KUKA KRL program: MyProgram_262().src

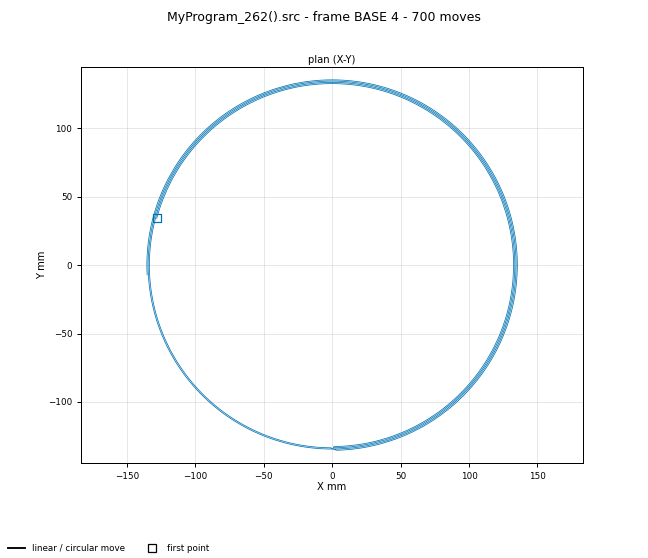
[picture p0: tool path of MyProgram_262().src in frame BASE 4, 700 of 700 moves have a stored position in this frame; points joined in program order, loops and branches not executed]
&ACCESS RVP
&REL 1
&PARAM TEMPLATE = C:\KRC\Roboter\Template\vorgabe
&PARAM EDITMASK = *
DEF MyProgram_262()
; ---- Setting reference (Base) ----
$BASE = BASE_DATA[4]

; --------------------------
; ---- Setting tool (TCP) ----
$TOOL = TOOL_DATA[3]
; --------------------------

$VEL.CP = VEL_APROX_PRINT
Startdeposition()
$VEL.CP = VEL_PRINT
LIN {X -128.1106,Y 34.116,Z 168,A 165.358,B 10.6516,C 0.1235,E1 10.4979,E2 285.5188} C_DIS
LIN {X -127.1106,Y 37.6736,Z 168,A 163.7129,B 10.6516,C 0.1199,E1 10.4991,E2 287.1678} C_DIS
LIN {X -125.942,Y 41.4132,Z 168,A 161.9508,B 10.6516,C 0.1164,E1 10.5006,E2 288.9361} C_DIS
LIN {X -124.5968,Y 45.2984,Z 168,A 160.2681,B 10.6518,C 0.1097,E1 10.5022,E2 290.6058} C_DIS
LIN {X -123.3963,Y 48.4742,Z 168,A 158.6213,B 10.6518,C 0.109,E1 10.5039,E2 292.272} C_DIS
LIN {X -120.4612,Y 55.3657,Z 168,A 155.2422,B 10.6518,C 0.1029,E1 10.5077,E2 295.6641} C_DIS
LIN {X -117.7741,Y 60.8777,Z 168,A 152.6518,B 10.6518,C 0.0948,E1 10.5109,E2 298.2447} C_DIS
LIN {X -115.8376,Y 64.4859,Z 168,A 150.9654,B 10.6519,C 0.0886,E1 10.5131,E2 299.9194} C_DIS
LIN {X -113.7435,Y 68.1115,Z 168,A 149.1743,B 10.6519,C 0.0836,E1 10.5157,E2 301.7063} C_DIS
LIN {X -110.9155,Y 72.626,Z 168,A 147.0442,B 10.6521,C 0.0746,E1 10.5188,E2 303.8138} C_DIS
LIN {X -109.3081,Y 75.0228,Z 168,A 145.5131,B 10.6521,C 0.0769,E1 10.5213,E2 305.3767} C_DIS
LIN {X -106.8216,Y 78.5228,Z 168,A 143.6005,B 10.6521,C 0.0735,E1 10.5244,E2 307.294} C_DIS
LIN {X -104.1665,Y 82.0125,Z 168,A 141.7197,B 10.6521,C 0.0688,E1 10.5276,E2 309.1711} C_DIS
LIN {X -101.3729,Y 85.4419,Z 168,A 139.7836,B 10.6521,C 0.0649,E1 10.531,E2 311.1079} C_DIS
LIN {X -98.5887,Y 88.6398,Z 168,A 137.9057,B 10.6521,C 0.0617,E1 10.5345,E2 312.9892} C_DIS
LIN {X -95.5472,Y 91.9108,Z 168,A 135.9314,B 10.6521,C 0.0583,E1 10.5383,E2 314.9666} C_DIS
LIN {X -92.4629,Y 95.0127,Z 168,A 134.0224,B 10.6521,C 0.0547,E1 10.5421,E2 316.8759} C_DIS
LIN {X -89.2719,Y 98.0167,Z 168,A 132.1098,B 10.6521,C 0.0512,E1 10.546,E2 318.7886} C_DIS
LIN {X -86.0227,Y 100.8802,Z 168,A 130.2329,B 10.6522,C 0.0477,E1 10.55,E2 320.6642} C_DIS
LIN {X -82.589,Y 103.7099,Z 168,A 128.2998,B 10.6522,C 0.0443,E1 10.5542,E2 322.5966} C_DIS
LIN {X -79.0187,Y 106.4555,Z 168,A 126.3454,B 10.6522,C 0.0409,E1 10.5585,E2 324.55} C_DIS
LIN {X -75.68,Y 108.8542,Z 168,A 124.5397,B 10.6522,C 0.0384,E1 10.5626,E2 326.3574} C_DIS
LIN {X -72.0548,Y 111.2871,Z 168,A 122.6403,B 10.6522,C 0.0355,E1 10.5671,E2 328.2565} C_DIS
LIN {X -68.5115,Y 113.5028,Z 168,A 120.4154,B 10.6522,C 0.041,E1 10.5725,E2 330.5284} C_DIS
LIN {X -64.82,Y 115.6507,Z 168,A 118.4323,B 10.6522,C 0.041,E1 10.5774,E2 332.5256} C_DIS
LIN {X -60.5627,Y 117.9344,Z 168,A 117.1036,B 10.6522,C 0.0229,E1 10.5804,E2 333.7644} C_DIS
LIN {X -53.8546,Y 121.1443,Z 168,A 113.7444,B 10.6522,C 0.0217,E1 10.589,E2 337.1379} C_DIS
LIN {X -50.7874,Y 122.4619,Z 168,A 112.2996,B 10.6522,C 0.02,E1 10.5927,E2 338.5818} C_DIS
LIN {X -47.6217,Y 123.7277,Z 168,A 110.7107,B 10.6522,C 0.0207,E1 10.5968,E2 340.183} C_DIS
LIN {X -43.62,Y 125.194,Z 168,A 108.8903,B 10.6522,C 0.0184,E1 10.6016,E2 341.9994} C_DIS
LIN {X -37.8929,Y 127.0464,Z 168,A 106.3941,B 10.6523,C 0.0138,E1 10.6082,E2 344.4815} C_DIS
LIN {X -34.225,Y 128.0815,Z 168,A 104.6813,B 10.6523,C 0.0138,E1 10.6128,E2 346.2008} C_DIS
LIN {X -31.0238,Y 128.8943,Z 168,A 102.7778,B 10.6523,C 0.0227,E1 10.6181,E2 348.1586} C_DIS
LIN {X -26.9831,Y 129.8016,Z 168,A 101.3362,B 10.6523,C 0.0143,E1 10.622,E2 349.5587} C_DIS
LIN {X -23.2949,Y 130.5128,Z 168,A 99.8078,B 10.6523,C 0.0113,E1 10.6261,E2 351.075} C_DIS
LIN {X -20.1004,Y 131.043,Z 168,A 98.4194,B 10.6523,C 0.0104,E1 10.63,E2 352.4612} C_DIS
LIN {X -16.8033,Y 131.507,Z 168,A 96.8595,B 10.6523,C 0.0123,E1 10.6343,E2 354.0344} C_DIS
LIN {X -12.6917,Y 131.9667,Z 168,A 95.1681,B 10.6523,C 0.0096,E1 10.639,E2 355.7135} C_DIS
LIN {X -9.1067,Y 132.2636,Z 168,A 93.5018,B 10.6523,C 0.0116,E1 10.6436,E2 357.392} C_DIS
LIN {X -5.0768,Y 132.4784,Z 168,A 91.8892,B 10.6523,C 0.0085,E1 10.6481,E2 358.9883} C_DIS
LIN {X -1.0548,Y 132.5719,Z 168,A 90.0932,B 10.6523,C 0.0096,E1 10.6531,E2 360.7902} C_DIS
LIN {X 3.0141,Y 132.5431,Z 168,A 88.2853,B 10.6523,C 0.0106,E1 10.6582,E2 362.6032} C_DIS
LIN {X 6.8789,Y 132.3972,Z 168,A 86.621,B 10.6523,C 0.0106,E1 10.6628,E2 364.2659} C_DIS
LIN {X 11.0997,Y 132.1101,Z 168,A 84.8958,B 10.6523,C 0.0087,E1 10.6676,E2 365.9783} C_DIS
LIN {X 14.6757,Y 131.7617,Z 168,A 83.2175,B 10.6523,C 0.0118,E1 10.6723,E2 367.6707} C_DIS
LIN {X 18.6908,Y 131.2514,Z 168,A 81.5841,B 10.6523,C 0.0099,E1 10.6768,E2 369.29} C_DIS
LIN {X 22.2463,Y 130.6964,Z 168,A 79.9517,B 10.6523,C 0.0123,E1 10.6813,E2 370.931} C_DIS
LIN {X 26.3227,Y 129.936,Z 168,A 78.219,B 10.6523,C 0.0119,E1 10.686,E2 372.6562} C_DIS
LIN {X 29.724,Y 129.2005,Z 168,A 76.7426,B 10.6523,C 0.0121,E1 10.6901,E2 374.1291} C_DIS
LIN {X 33.368,Y 128.3098,Z 168,A 74.8518,B 10.6523,C 0.0193,E1 10.6953,E2 376.0512} C_DIS
LIN {X 38.226,Y 126.9462,Z 168,A 72.8076,B 10.6523,C 0.0179,E1 10.7007,E2 378.0791} C_DIS
LIN {X 41.8818,Y 125.786,Z 168,A 71.2962,B 10.6523,C 0.016,E1 10.7047,E2 379.5731} C_DIS
LIN {X 45.2416,Y 124.6173,Z 168,A 69.7429,B 10.6523,C 0.0178,E1 10.7088,E2 381.1281} C_DIS
LIN {X 49.8552,Y 122.8444,Z 168,A 67.6692,B 10.6523,C 0.0186,E1 10.7141,E2 383.1943} C_DIS
LIN {X 52.8378,Y 121.5911,Z 168,A 66.2142,B 10.6523,C 0.0214,E1 10.7179,E2 384.656} C_DIS
LIN {X 56.1015,Y 120.1209,Z 168,A 64.7425,B 10.6523,C 0.0215,E1 10.7216,E2 386.1189} C_DIS
LIN {X 59.3042,Y 118.5736,Z 168,A 63.1993,B 10.6523,C 0.0236,E1 10.7255,E2 387.6629} C_DIS
LIN {X 62.612,Y 116.8608,Z 168,A 61.5001,B 10.6523,C 0.0278,E1 10.7297,E2 389.3727} C_DIS
LIN {X 66.5457,Y 114.6664,Z 168,A 59.672,B 10.6523,C 0.0278,E1 10.7341,E2 391.187} C_DIS
LIN {X 69.8181,Y 112.704,Z 168,A 57.9049,B 10.6523,C 0.033,E1 10.7383,E2 392.9682} C_DIS
LIN {X 74.2551,Y 109.8311,Z 168,A 55.9079,B 10.6523,C 0.0298,E1 10.7429,E2 394.9318} C_DIS
LIN {X 76.5411,Y 108.2505,Z 168,A 54.5126,B 10.6523,C 0.0363,E1 10.7462,E2 396.3502} C_DIS
LIN {X 79.8218,Y 105.8544,Z 168,A 52.7643,B 10.6523,C 0.0392,E1 10.7501,E2 398.0981} C_DIS
LIN {X 83.4409,Y 103.0261,Z 168,A 51.0245,B 10.6523,C 0.0369,E1 10.7539,E2 399.8094} C_DIS
LIN {X 85.6135,Y 101.2281,Z 168,A 49.5107,B 10.6523,C 0.0461,E1 10.7572,E2 401.3584} C_DIS
LIN {X 89.0951,Y 98.1771,Z 168,A 47.5797,B 10.6523,C 0.0483,E1 10.7612,E2 403.2819} C_DIS
LIN {X 92.2102,Y 95.2573,Z 168,A 45.7442,B 10.6522,C 0.0517,E1 10.7649,E2 405.1168} C_DIS
LIN {X 95.4598,Y 92.0011,Z 168,A 43.7862,B 10.6522,C 0.0551,E1 10.7687,E2 407.072} C_DIS
LIN {X 98.4767,Y 88.7649,Z 168,A 41.8428,B 10.6522,C 0.0599,E1 10.7724,E2 409.02} C_DIS
LIN {X 101.386,Y 85.4262,Z 168,A 39.6499,B 10.6521,C 0.0708,E1 10.7764,E2 411.2467} C_DIS
LIN {X 103.8717,Y 82.3857,Z 168,A 38.5136,B 10.6521,C 0.061,E1 10.7783,E2 412.3176} C_DIS
LIN {X 106.0357,Y 79.5816,Z 168,A 36.7864,B 10.6521,C 0.0693,E1 10.7813,E2 414.0689} C_DIS
LIN {X 109.0261,Y 75.4329,Z 168,A 34.5872,B 10.6521,C 0.0743,E1 10.7848,E2 416.268} C_DIS
LIN {X 111.473,Y 71.7675,Z 168,A 32.7191,B 10.6521,C 0.078,E1 10.7877,E2 418.1329} C_DIS
LIN {X 114.9912,Y 65.9835,Z 168,A 29.9104,B 10.652,C 0.0824,E1 10.7917,E2 420.9295} C_DIS
LIN {X 116.7459,Y 62.826,Z 168,A 28.305,B 10.652,C 0.0874,E1 10.7938,E2 422.5412} C_DIS
LIN {X 119.2337,Y 57.9661,Z 168,A 26.0578,B 10.652,C 0.0907,E1 10.7966,E2 424.7767} C_DIS
LIN {X 120.55,Y 55.1737,Z 168,A 24.7613,B 10.652,C 0.0933,E1 10.7982,E2 426.0697} C_DIS
LIN {X 121.9386,Y 52.0341,Z 168,A 23.0437,B 10.6518,C 0.1031,E1 10.8001,E2 427.8162} C_DIS
LIN {X 123.5333,Y 48.1218,Z 168,A 21.452,B 10.6518,C 0.1022,E1 10.8017,E2 429.3814} C_DIS
LIN {X 124.9473,Y 44.3264,Z 168,A 19.5951,B 10.6518,C 0.1096,E1 10.8035,E2 431.2524} C_DIS
LIN {X 127.0875,Y 37.7525,Z 168,A 16.9155,B 10.6518,C 0.1102,E1 10.8058,E2 433.8976} C_DIS
LIN {X 127.971,Y 34.6393,Z 168,A 15.5452,B 10.6518,C 0.1134,E1 10.8068,E2 435.2658} C_DIS
LIN {X 128.8941,Y 31.0247,Z 168,A 13.8162,B 10.6516,C 0.1209,E1 10.808,E2 437.0101} C_DIS
LIN {X 129.5973,Y 27.9424,Z 168,A 12.4748,B 10.6516,C 0.1242,E1 10.8088,E2 438.3498} C_DIS
LIN {X 130.2591,Y 24.6751,Z 168,A 10.9452,B 10.6516,C 0.1305,E1 10.8096,E2 439.8913} C_DIS
LIN {X 131.0119,Y 20.301,Z 168,A 9.1266,B 10.6515,C 0.1335,E1 10.8104,E2 441.6997} C_DIS
LIN {X 131.6021,Y 16.0401,Z 168,A 7.2764,B 10.6515,C 0.1387,E1 10.8111,E2 443.5506} C_DIS
LIN {X 131.9953,Y 12.3938,Z 168,A 5.6463,B 10.6513,C 0.1445,E1 10.8115,E2 445.1877} C_DIS
LIN {X 132.3248,Y 8.1515,Z 168,A 3.9615,B 10.6513,C 0.1459,E1 10.8119,E2 446.8558} C_DIS
LIN {X 132.5061,Y 4.3453,Z 168,A 2.2154,B 10.6513,C 0.1533,E1 10.8121,E2 448.6155} C_DIS
LIN {X 132.5788,Y 0.1484,Z 168,A 0.4111,B 10.6511,C 0.1584,E1 10.8121,E2 450.4205} C_DIS
LIN {X 132.5201,Y -3.8421,Z 168,A -1.1832,B 10.6511,C 0.1601,E1 10.8121,E2 452.0008} C_DIS
LIN {X 132.2957,Y -8.6229,Z 168,A -3.1135,B 10.6511,C 0.1627,E1 10.8117,E2 453.9167} C_DIS
LIN {X 132.0836,Y -11.4138,Z 168,A -4.3432,B 10.6511,C 0.1667,E1 10.8115,E2 455.15} C_DIS
LIN {X 131.8176,Y -14.1563,Z 168,A -5.6008,B 10.6509,C 0.1719,E1 10.8111,E2 456.4169} C_DIS
LIN {X 131.4241,Y -17.4363,Z 168,A -6.9971,B 10.6509,C 0.1753,E1 10.8106,E2 457.811} C_DIS
LIN {X 130.9027,Y -21.0067,Z 168,A -8.65,B 10.6508,C 0.1822,E1 10.8099,E2 459.4769} C_DIS
LIN {X 130.2276,Y -24.8401,Z 168,A -10.2162,B 10.6508,C 0.1841,E1 10.8091,E2 461.0308} C_DIS
LIN {X 129.5629,Y -28.1016,Z 168,A -12.0731,B 10.6505,C 0.1988,E1 10.808,E2 462.9396} C_DIS
LIN {X 128.5971,Y -32.2361,Z 168,A -13.494,B 10.6505,C 0.1937,E1 10.8071,E2 464.3129} C_DIS
LIN {X 127.6192,Y -35.9109,Z 168,A -15.0264,B 10.6505,C 0.1956,E1 10.806,E2 465.8336} C_DIS
LIN {X 126.581,Y -39.4191,Z 168,A -16.8727,B 10.6503,C 0.2068,E1 10.8044,E2 467.7136} C_DIS
LIN {X 124.9719,Y -44.2582,Z 168,A -18.7569,B 10.6503,C 0.2049,E1 10.8027,E2 469.5618} C_DIS
LIN {X 123.6627,Y -47.789,Z 168,A -20.4493,B 10.6503,C 0.211,E1 10.8011,E2 471.2638} C_DIS
LIN {X 122.2513,Y -51.2917,Z 168,A -21.9706,B 10.6503,C 0.2127,E1 10.7995,E2 472.7735} C_DIS
LIN {X 120.7627,Y -54.7077,Z 168,A -24.4708,B 10.6497,C 0.2394,E1 10.7965,E2 475.3823} C_DIS
LIN {X 117.9763,Y -60.4805,Z 168,A -26.4123,B 10.6499,C 0.2261,E1 10.7941,E2 477.2276} C_DIS
LIN {X 115.6389,Y -64.841,Z 168,A -28.4716,B 10.6499,C 0.2298,E1 10.7914,E2 479.2799} C_DIS
LIN {X 113.5551,Y -68.4249,Z 168,A -30.2759,B 10.6498,C 0.2347,E1 10.7888,E2 481.0877} C_DIS
LIN {X 111.358,Y -71.9456,Z 168,A -32.0094,B 10.6497,C 0.2378,E1 10.7862,E2 482.816} C_DIS
LIN {X 109.0382,Y -75.4155,Z 168,A -33.8717,B 10.6496,C 0.2437,E1 10.7833,E2 484.6873} C_DIS
LIN {X 106.4297,Y -79.0533,Z 168,A -35.7464,B 10.6495,C 0.2469,E1 10.7802,E2 486.5569} C_DIS
LIN {X 103.6859,Y -82.6192,Z 168,A -37.7453,B 10.6493,C 0.2529,E1 10.7768,E2 488.5645} C_DIS
LIN {X 101.0311,Y -85.8453,Z 168,A -39.2495,B 10.6494,C 0.2496,E1 10.7741,E2 490.0341} C_DIS
LIN {X 98.7917,Y -88.4132,Z 168,A -40.9101,B 10.6492,C 0.2576,E1 10.771,E2 491.7191} C_DIS
LIN {X 95.6925,Y -91.7588,Z 168,A -42.9523,B 10.6491,C 0.2637,E1 10.7671,E2 493.772} C_DIS
LIN {X 91.9906,Y -95.47,Z 168,A -45.0402,B 10.6491,C 0.2642,E1 10.763,E2 495.8408} C_DIS
LIN {X 89.1014,Y -98.1714,Z 168,A -46.7684,B 10.649,C 0.2682,E1 10.7594,E2 497.573} C_DIS
LIN {X 85.8546,Y -101.0232,Z 168,A -48.7195,B 10.6488,C 0.274,E1 10.7553,E2 499.5362} C_DIS
LIN {X 82.5788,Y -103.718,Z 168,A -50.4228,B 10.6488,C 0.2744,E1 10.7516,E2 501.2256} C_DIS
LIN {X 79.3579,Y -106.2029,Z 168,A -52.1823,B 10.6488,C 0.2777,E1 10.7477,E2 502.9871} C_DIS
LIN {X 76.0244,Y -108.6146,Z 168,A -53.9904,B 10.6486,C 0.2817,E1 10.7436,E2 504.8005} C_DIS
LIN {X 71.7145,Y -111.507,Z 168,A -56.0496,B 10.6486,C 0.2811,E1 10.7388,E2 506.8395} C_DIS
LIN {X 68.5128,Y -113.502,Z 168,A -57.8012,B 10.6485,C 0.2867,E1 10.7346,E2 508.6074} C_DIS
LIN {X 64.9262,Y -115.591,Z 168,A -59.5239,B 10.6485,C 0.2878,E1 10.7304,E2 510.323} C_DIS
LIN {X 61.3961,Y -117.5021,Z 168,A -61.2539,B 10.6485,C 0.2902,E1 10.7262,E2 512.054} C_DIS
LIN {X 58.289,Y -119.0744,Z 168,A -62.7276,B 10.6484,C 0.2916,E1 10.7225,E2 513.5253} C_DIS
LIN {X 54.8872,Y -120.6822,Z 168,A -64.5319,B 10.6482,C 0.2981,E1 10.7179,E2 515.3526} C_DIS
LIN {X 50.9136,Y -122.4092,Z 168,A -66.2028,B 10.6482,C 0.2956,E1 10.7136,E2 517.0005} C_DIS
LIN {X 47.6548,Y -123.7149,Z 168,A -67.7073,B 10.6482,C 0.2972,E1 10.7097,E2 518.5048} C_DIS
LIN {X 44.3277,Y -124.9468,Z 168,A -69.5932,B 10.6479,C 0.3071,E1 10.7046,E2 520.4346} C_DIS
LIN {X 40.9009,Y -126.1097,Z 168,A -70.6744,B 10.6482,C 0.2975,E1 10.7019,E2 521.4586} C_DIS
LIN {X 34.9271,Y -127.894,Z 168,A -73.7797,B 10.6479,C 0.3096,E1 10.6935,E2 524.6157} C_DIS
LIN {X 31.6962,Y -128.7323,Z 168,A -74.8167,B 10.6481,C 0.3014,E1 10.6908,E2 525.6046} C_DIS
LIN {X 27.0777,Y -129.7824,Z 168,A -77.0733,B 10.6479,C 0.3078,E1 10.6846,E2 527.888} C_DIS
LIN {X 23.1472,Y -130.5393,Z 168,A -78.6722,B 10.6479,C 0.3059,E1 10.6802,E2 529.4721} C_DIS
LIN {X 19.6209,Y -131.1172,Z 168,A -80.3073,B 10.6479,C 0.3089,E1 10.6757,E2 531.1193} C_DIS
LIN {X 15.7765,Y -131.6335,Z 168,A -81.8945,B 10.6479,C 0.3077,E1 10.6713,E2 532.6966} C_DIS
LIN {X 12.6831,Y -131.9675,Z 168,A -83.2375,B 10.6479,C 0.3082,E1 10.6676,E2 534.0401} C_DIS
LIN {X 8.8727,Y -132.2804,Z 168,A -84.9306,B 10.6479,C 0.3097,E1 10.6628,E2 535.7392} C_DIS
LIN {X 5.1248,Y -132.4766,Z 168,A -86.4825,B 10.6479,C 0.3086,E1 10.6585,E2 537.2834} C_DIS
LIN {X 1.4089,Y -132.57,Z 168,A -88.2295,B 10.6478,C 0.312,E1 10.6536,E2 539.0482} C_DIS
LIN {X 1.4089,Y -132.57,Z 168,A -88.2295,B 10.6478,C 0.312,E1 10.6536,E2 539.0482} C_DIS
Enddeposition()
LIN {X 0.9669,Y -133.4849,Z 168,A -87.6849,B 10.648,C 0.3018,E1 10.6552,E2 538.4484} C_DIS
Startdeposition()
$VEL.CP = VEL_PRINT
LIN {X 4.8347,Y -133.4026,Z 168,A -85.925,B 10.6481,C 0.2991,E1 10.6602,E2 536.6754} C_DIS
LIN {X 8.3118,Y -133.2306,Z 168,A -84.4038,B 10.6481,C 0.2981,E1 10.6644,E2 535.15} C_DIS
LIN {X 12.5232,Y -132.901,Z 168,A -82.606,B 10.6481,C 0.2977,E1 10.6694,E2 533.3531} C_DIS
LIN {X 16.497,Y -132.468,Z 168,A -80.8583,B 10.6481,C 0.2962,E1 10.6743,E2 531.6005} C_DIS
LIN {X 20.1133,Y -131.9659,Z 168,A -79.348,B 10.6481,C 0.2967,E1 10.6784,E2 530.0962} C_DIS
LIN {X 23.4585,Y -131.4121,Z 168,A -77.8636,B 10.6482,C 0.2951,E1 10.6825,E2 528.6073} C_DIS
LIN {X 27.714,Y -130.5816,Z 168,A -76.0404,B 10.6482,C 0.2946,E1 10.6875,E2 526.7875} C_DIS
LIN {X 31.227,Y -129.7855,Z 168,A -74.7322,B 10.6482,C 0.299,E1 10.691,E2 525.5076} C_DIS
LIN {X 38.5059,Y -127.8164,Z 168,A -71.3936,B 10.6482,C 0.2938,E1 10.7,E2 522.1544} C_DIS
LIN {X 44.7941,Y -125.7502,Z 168,A -68.4105,B 10.6484,C 0.2874,E1 10.708,E2 519.1517} C_DIS
LIN {X 48.32,Y -124.4369,Z 168,A -66.8821,B 10.6484,C 0.2876,E1 10.7119,E2 517.6326} C_DIS
LIN {X 51.0917,Y -123.3253,Z 168,A -65.436,B 10.6486,C 0.282,E1 10.7157,E2 516.1651} C_DIS
LIN {X 55.6069,Y -121.3566,Z 168,A -63.4435,B 10.6486,C 0.2822,E1 10.7208,E2 514.186} C_DIS
LIN {X 59.0659,Y -119.7103,Z 168,A -61.8408,B 10.6486,C 0.2809,E1 10.7248,E2 512.5869} C_DIS
LIN {X 62.1173,Y -118.1557,Z 168,A -60.415,B 10.6486,C 0.2799,E1 10.7283,E2 511.1653} C_DIS
LIN {X 65.4631,Y -116.3377,Z 168,A -58.7385,B 10.6487,C 0.2764,E1 10.7324,E2 509.4821} C_DIS
LIN {X 68.8897,Y -114.3422,Z 168,A -56.9772,B 10.6488,C 0.2722,E1 10.7367,E2 507.7119} C_DIS
LIN {X 75.2735,Y -110.2446,Z 168,A -53.7623,B 10.6489,C 0.2677,E1 10.7442,E2 504.4991} C_DIS
LIN {X 78.748,Y -107.7903,Z 168,A -51.9302,B 10.649,C 0.2642,E1 10.7483,E2 502.6644} C_DIS
LIN {X 81.2992,Y -105.8791,Z 168,A -50.4601,B 10.6491,C 0.2591,E1 10.7516,E2 501.1804} C_DIS
LIN {X 86.9331,Y -101.3043,Z 168,A -47.4994,B 10.6491,C 0.2568,E1 10.758,E2 498.2356} C_DIS
LIN {X 90.0179,Y -98.574,Z 168,A -45.6993,B 10.6493,C 0.2524,E1 10.7617,E2 496.4298} C_DIS
LIN {X 93.429,Y -95.3462,Z 168,A -43.3496,B 10.6496,C 0.2397,E1 10.7665,E2 494.0363} C_DIS
LIN {X 96.4916,Y -92.2456,Z 168,A -41.9245,B 10.6494,C 0.2468,E1 10.7692,E2 492.6647} C_DIS
LIN {X 99.5283,Y -88.9607,Z 168,A -40.1408,B 10.6494,C 0.246,E1 10.7725,E2 490.8959} C_DIS
LIN {X 101.6026,Y -86.584,Z 168,A -38.2766,B 10.6498,C 0.2299,E1 10.776,E2 488.9668} C_DIS
LIN {X 104.3253,Y -83.2835,Z 168,A -36.8372,B 10.6497,C 0.2357,E1 10.7784,E2 487.5748} C_DIS
LIN {X 107.1524,Y -79.6131,Z 168,A -34.9386,B 10.6497,C 0.2332,E1 10.7816,E2 485.6852} C_DIS
LIN {X 109.6238,Y -76.1741,Z 168,A -33.1093,B 10.6498,C 0.2284,E1 10.7846,E2 483.8524} C_DIS
LIN {X 112.1361,Y -72.4256,Z 168,A -31.1662,B 10.6499,C 0.2234,E1 10.7876,E2 481.9065} C_DIS
LIN {X 114.3136,Y -68.937,Z 168,A -29.4994,B 10.6499,C 0.2214,E1 10.79,E2 480.2499} C_DIS
LIN {X 116.2062,Y -65.697,Z 168,A -27.8161,B 10.6501,C 0.2153,E1 10.7923,E2 478.5557} C_DIS
LIN {X 118.2765,Y -61.8873,Z 168,A -26.0484,B 10.6501,C 0.2128,E1 10.7946,E2 476.7974} C_DIS
LIN {X 120.9198,Y -56.5482,Z 168,A -23.4234,B 10.6503,C 0.2042,E1 10.7978,E2 474.1612} C_DIS
LIN {X 122.8642,Y -52.1958,Z 168,A -21.4179,B 10.6504,C 0.1997,E1 10.8001,E2 472.1585} C_DIS
LIN {X 124.2594,Y -48.7767,Z 168,A -19.7831,B 10.6505,C 0.194,E1 10.8018,E2 470.5158} C_DIS
LIN {X 126.1727,Y -43.5873,Z 168,A -17.002,B 10.6508,C 0.1768,E1 10.8044,E2 467.6813} C_DIS
LIN {X 127.7609,Y -38.6872,Z 168,A -15.7921,B 10.6505,C 0.1964,E1 10.8053,E2 466.5929} C_DIS
LIN {X 128.6735,Y -35.5348,Z 168,A -13.5132,B 10.6509,C 0.1699,E1 10.8071,E2 464.205} C_DIS
LIN {X 129.8359,Y -31.018,Z 168,A -12.0404,B 10.6508,C 0.1779,E1 10.808,E2 462.7956} C_DIS
LIN {X 130.7522,Y -26.8952,Z 168,A -10.3023,B 10.6508,C 0.1746,E1 10.809,E2 461.0647} C_DIS
LIN {X 131.3953,Y -23.5524,Z 168,A -8.8754,B 10.6508,C 0.1712,E1 10.8098,E2 459.6404} C_DIS
LIN {X 131.971,Y -20.0805,Z 168,A -7.2524,B 10.651,C 0.1639,E1 10.8105,E2 458.0019} C_DIS
LIN {X 132.5251,Y -16.0184,Z 168,A -5.6064,B 10.651,C 0.1617,E1 10.8111,E2 456.368} C_DIS
LIN {X 132.9538,Y -11.9699,Z 168,A -3.8108,B 10.6511,C 0.1554,E1 10.8115,E2 454.5648} C_DIS
LIN {X 133.3795,Y -5.4277,Z 168,A -1.1016,B 10.6512,C 0.1498,E1 10.812,E2 451.8655} C_DIS
LIN {X 133.4828,Y -1.5221,Z 168,A 0.5483,B 10.6512,C 0.1456,E1 10.812,E2 450.2172} C_DIS
LIN {X 133.4659,Y 2.5399,Z 168,A 2.3503,B 10.6514,C 0.139,E1 10.812,E2 448.4063} C_DIS
LIN {X 133.3293,Y 6.5422,Z 168,A 3.9564,B 10.6514,C 0.1368,E1 10.8118,E2 446.8123} C_DIS
LIN {X 133.0687,Y 10.6103,Z 168,A 5.7499,B 10.6514,C 0.1306,E1 10.8114,E2 445.0117} C_DIS
LIN {X 132.7083,Y 14.422,Z 168,A 7.2979,B 10.6514,C 0.1283,E1 10.811,E2 443.4737} C_DIS
LIN {X 132.2159,Y 18.4024,Z 168,A 9.029,B 10.6516,C 0.123,E1 10.8104,E2 441.7399} C_DIS
LIN {X 131.6516,Y 22.0751,Z 168,A 10.5384,B 10.6516,C 0.1206,E1 10.8097,E2 440.2395} C_DIS
LIN {X 130.9528,Y 25.9094,Z 168,A 12.3184,B 10.6516,C 0.1131,E1 10.8088,E2 438.4449} C_DIS
LIN {X 130.1492,Y 29.6751,Z 168,A 13.8629,B 10.6516,C 0.1111,E1 10.8078,E2 436.9121} C_DIS
LIN {X 129.143,Y 33.7917,Z 168,A 15.5266,B 10.6516,C 0.11,E1 10.8067,E2 435.2658} C_DIS
LIN {X 128.1592,Y 37.345,Z 168,A 17.4715,B 10.6518,C 0.0963,E1 10.8052,E2 433.2753} C_DIS
LIN {X 127.2033,Y 40.4812,Z 168,A 18.7798,B 10.6518,C 0.0949,E1 10.8041,E2 431.9779} C_DIS
LIN {X 125.6983,Y 44.938,Z 168,A 20.5547,B 10.6518,C 0.0956,E1 10.8025,E2 430.2312} C_DIS
LIN {X 123.4553,Y 50.7801,Z 168,A 23.239,B 10.6518,C 0.0884,E1 10.7998,E2 427.5451} C_DIS
LIN {X 122.0547,Y 54.0576,Z 168,A 24.7465,B 10.6519,C 0.0849,E1 10.7981,E2 426.0392} C_DIS
LIN {X 120.5533,Y 57.3262,Z 168,A 26.1588,B 10.6519,C 0.0841,E1 10.7964,E2 424.6417} C_DIS
LIN {X 117.8281,Y 62.7412,Z 168,A 30.0013,B 10.6522,C 0.046,E1 10.7912,E2 420.6453} C_DIS
LIN {X 113.8573,Y 69.6879,Z 168,A 32.2961,B 10.6521,C 0.0663,E1 10.7882,E2 418.4885} C_DIS
LIN {X 111.4042,Y 73.5459,Z 168,A 34.2452,B 10.6521,C 0.0619,E1 10.7852,E2 416.5397} C_DIS
LIN {X 109.7454,Y 75.9994,Z 168,A 35.9748,B 10.6521,C 0.0474,E1 10.7824,E2 414.7537} C_DIS
LIN {X 106.9923,Y 79.8282,Z 168,A 38.3304,B 10.6522,C 0.0344,E1 10.7783,E2 412.3563} C_DIS
LIN {X 102.9133,Y 85.022,Z 168,A 40.3008,B 10.6522,C 0.0497,E1 10.775,E2 410.4901} C_DIS
LIN {X 100.0268,Y 88.3997,Z 168,A 42.1611,B 10.6522,C 0.0467,E1 10.7716,E2 408.6347} C_DIS
LIN {X 97.1384,Y 91.5642,Z 168,A 44.0074,B 10.6522,C 0.0426,E1 10.7681,E2 406.7867} C_DIS
LIN {X 93.9942,Y 94.7891,Z 168,A 45.9057,B 10.6522,C 0.0395,E1 10.7644,E2 404.8919} C_DIS
LIN {X 90.7762,Y 97.8755,Z 168,A 47.8048,B 10.6522,C 0.0361,E1 10.7605,E2 402.9939} C_DIS
LIN {X 87.528,Y 100.791,Z 168,A 49.6881,B 10.6522,C 0.0323,E1 10.7566,E2 401.1088} C_DIS
LIN {X 84.1951,Y 103.5914,Z 168,A 51.9804,B 10.6522,C 0.0186,E1 10.7515,E2 398.7646} C_DIS
LIN {X 80.6051,Y 106.4084,Z 168,A 53.4903,B 10.6522,C 0.0261,E1 10.7483,E2 397.3086} C_DIS
LIN {X 77.6382,Y 108.5918,Z 168,A 55.5211,B 10.6522,C 0.0126,E1 10.7436,E2 395.2229} C_DIS
LIN {X 73.7147,Y 111.2931,Z 168,A 57.1059,B 10.6522,C 0.0204,E1 10.74,E2 393.6935} C_DIS
LIN {X 70.0596,Y 113.6293,Z 168,A 58.9354,B 10.6522,C 0.0184,E1 10.7357,E2 391.8677} C_DIS
LIN {X 64.2417,Y 117.0171,Z 168,A 61.8156,B 10.6522,C 0.0146,E1 10.7287,E2 388.9884} C_DIS
LIN {X 61.3529,Y 118.5571,Z 168,A 63.3181,B 10.6522,C 0.0104,E1 10.7249,E2 387.4741} C_DIS
LIN {X 57.2842,Y 120.5734,Z 168,A 65.0699,B 10.6522,C 0.0127,E1 10.7206,E2 385.7459} C_DIS
LIN {X 53.3063,Y 122.3843,Z 168,A 66.8836,B 10.6522,C 0.012,E1 10.716,E2 383.9397} C_DIS
LIN {X 50.3075,Y 123.6475,Z 168,A 68.5495,B 10.6522,C 0.0042,E1 10.7116,E2 382.2415} C_DIS
LIN {X 45.5315,Y 125.4844,Z 168,A 70.5119,B 10.6522,C 0.0075,E1 10.7065,E2 380.3074} C_DIS
LIN {X 41.991,Y 126.7129,Z 168,A 72.3712,B 10.6522,C 0.0002,E1 10.7015,E2 378.4181} C_DIS
LIN {X 38.8564,Y 127.7091,Z 168,A 73.844,B 10.6522,C -0.0023,E1 10.6976,E2 376.9382} C_DIS
LIN {X 35.2378,Y 128.7565,Z 168,A 75.2233,B 10.6522,C 0.002,E1 10.6939,E2 375.5878} C_DIS
LIN {X 31.3751,Y 129.7498,Z 168,A 76.7729,B 10.6522,C 0.0045,E1 10.6898,E2 374.0579} C_DIS
LIN {X 28.3636,Y 130.4414,Z 168,A 78.1443,B 10.6522,C 0.0027,E1 10.6861,E2 372.6815} C_DIS
LIN {X 25.0098,Y 131.1256,Z 168,A 79.5885,B 10.6522,C 0.0025,E1 10.6821,E2 371.2406} C_DIS
LIN {X 21.2847,Y 131.7834,Z 168,A 81.2939,B 10.6522,C 0,E1 10.6774,E2 369.526} C_DIS
LIN {X 17.4857,Y 132.3394,Z 168,A 82.8428,B 10.6522,C 0.0016,E1 10.6731,E2 367.9893} C_DIS
LIN {X 14.1824,Y 132.734,Z 168,A 84.2815,B 10.6522,C 0.0009,E1 10.6691,E2 366.5498} C_DIS
LIN {X 10.0261,Y 133.1129,Z 168,A 86.0876,B 10.6522,C 0.0003,E1 10.6641,E2 364.7428} C_DIS
LIN {X 6.3405,Y 133.3395,Z 168,A 87.7434,B 10.6522,C -0.0015,E1 10.6595,E2 363.0792} C_DIS
LIN {X 2.1303,Y 133.4727,Z 168,A 89.4973,B 10.6522,C -0.0003,E1 10.6546,E2 361.3325} C_DIS
LIN {X -2.1618,Y 133.4722,Z 168,A 91.2998,B 10.6522,C 0.0007,E1 10.6496,E2 359.5355} C_DIS
LIN {X -6.1396,Y 133.3496,Z 168,A 93.0393,B 10.6522,C 0.0002,E1 10.6447,E2 357.7932} C_DIS
LIN {X -9.749,Y 133.1331,Z 168,A 94.6278,B 10.6522,C -0.0002,E1 10.6403,E2 356.2012} C_DIS
LIN {X -14.0786,Y 132.7452,Z 168,A 96.4588,B 10.6522,C 0.0012,E1 10.6352,E2 354.3753} C_DIS
LIN {X -18.1111,Y 132.2574,Z 168,A 98.2405,B 10.6522,C 0.0011,E1 10.6303,E2 352.5902} C_DIS
LIN {X -21.8348,Y 131.6917,Z 168,A 99.8071,B 10.6522,C 0.003,E1 10.626,E2 351.0305} C_DIS
LIN {X -25.3257,Y 131.0653,Z 168,A 101.3046,B 10.6522,C 0.0044,E1 10.6219,E2 349.5368} C_DIS
LIN {X -34.2827,Y 129.0121,Z 168,A 104.9997,B 10.6522,C 0.0126,E1 10.6119,E2 345.8743} C_DIS
LIN {X -41.7046,Y 126.8083,Z 168,A 108.5818,B 10.6522,C 0.0101,E1 10.6023,E2 342.2643} C_DIS
LIN {X -45.77,Y 125.3984,Z 168,A 110.5774,B 10.6522,C 0.0089,E1 10.5969,E2 340.2524} C_DIS
LIN {X -49.5704,Y 123.9446,Z 168,A 112.1958,B 10.6522,C 0.0135,E1 10.5928,E2 338.6506} C_DIS
LIN {X -52.9063,Y 122.5573,Z 168,A 113.8375,B 10.6522,C 0.0135,E1 10.5885,E2 336.9993} C_DIS
LIN {X -57.2463,Y 120.5915,Z 168,A 115.8891,B 10.6522,C 0.0159,E1 10.5833,E2 334.9487} C_DIS
LIN {X -60.124,Y 119.1834,Z 168,A 117.8466,B 10.6522,C 0.0057,E1 10.5783,E2 332.9227} C_DIS
LIN {X -64.4624,Y 116.8944,Z 168,A 119.446,B 10.6522,C 0.0192,E1 10.5745,E2 331.3859} C_DIS
LIN {X -68.4678,Y 114.5952,Z 168,A 121.4284,B 10.6522,C 0.0222,E1 10.5697,E2 329.4053} C_DIS
LIN {X -72.1984,Y 112.2824,Z 168,A 123.3126,B 10.6522,C 0.0252,E1 10.5653,E2 327.5228} C_DIS
LIN {X -75.7847,Y 109.8938,Z 168,A 125.1789,B 10.6522,C 0.028,E1 10.561,E2 325.6563} C_DIS
LIN {X -79.2891,Y 107.3928,Z 168,A 127.0912,B 10.6522,C 0.03,E1 10.5566,E2 323.7381} C_DIS
LIN {X -82.8508,Y 104.6697,Z 168,A 129.0521,B 10.6522,C 0.0328,E1 10.5523,E2 321.7747} C_DIS
LIN {X -86.3823,Y 101.7742,Z 168,A 130.991,B 10.6522,C 0.0369,E1 10.5482,E2 319.8403} C_DIS
LIN {X -89.8571,Y 98.7199,Z 168,A 132.9913,B 10.6522,C 0.0406,E1 10.544,E2 317.8402} C_DIS
LIN {X -93.094,Y 95.6739,Z 168,A 134.931,B 10.6522,C 0.0439,E1 10.5401,E2 315.8988} C_DIS
LIN {X -96.2393,Y 92.5095,Z 168,A 136.9029,B 10.6522,C 0.0469,E1 10.5362,E2 313.9221} C_DIS
LIN {X -99.3216,Y 89.1915,Z 168,A 138.8326,B 10.6522,C 0.0514,E1 10.5326,E2 311.996} C_DIS
LIN {X -102.3132,Y 85.7431,Z 168,A 140.7863,B 10.6522,C 0.056,E1 10.5291,E2 310.0452} C_DIS
LIN {X -105.094,Y 82.3113,Z 168,A 142.7106,B 10.6521,C 0.0598,E1 10.5257,E2 308.1195} C_DIS
LIN {X -107.7091,Y 78.8585,Z 168,A 144.6047,B 10.6521,C 0.0636,E1 10.5226,E2 306.2232} C_DIS
LIN {X -110.2018,Y 75.3358,Z 168,A 146.4806,B 10.6521,C 0.0676,E1 10.5196,E2 304.3465} C_DIS
LIN {X -111.8126,Y 72.9239,Z 168,A 148.1357,B 10.6521,C 0.0627,E1 10.517,E2 302.6436} C_DIS
LIN {X -114.0713,Y 69.3376,Z 168,A 149.6243,B 10.6521,C 0.0738,E1 10.5149,E2 301.1967} C_DIS
LIN {X -116.5003,Y 65.1738,Z 168,A 151.6487,B 10.652,C 0.08,E1 10.5121,E2 299.18} C_DIS
LIN {X -118.6135,Y 61.2434,Z 168,A 153.4906,B 10.652,C 0.0864,E1 10.5097,E2 297.349} C_DIS
LIN {X -120.1127,Y 58.245,Z 168,A 155.0333,B 10.6519,C 0.0882,E1 10.5078,E2 295.7954} C_DIS
LIN {X -121.3665,Y 55.5855,Z 168,A 156.3671,B 10.6519,C 0.0902,E1 10.5062,E2 294.4544} C_DIS
LIN {X -123.2819,Y 51.1957,Z 168,A 158.3553,B 10.6519,C 0.0971,E1 10.504,E2 292.4766} C_DIS
LIN {X -124.8565,Y 47.2272,Z 168,A 160.2141,B 10.6518,C 0.1017,E1 10.5022,E2 290.6167} C_DIS
LIN {X -126.1026,Y 43.7893,Z 168,A 161.8101,B 10.6518,C 0.1055,E1 10.5007,E2 289.0193} C_DIS
LIN {X -127.2139,Y 40.4479,Z 168,A 163.3766,B 10.6518,C 0.1087,E1 10.4993,E2 287.4478} C_DIS
LIN {X -128.4513,Y 36.3292,Z 168,A 165.2066,B 10.6517,C 0.1143,E1 10.4979,E2 285.6217} C_DIS
LIN {X -129.3712,Y 32.9012,Z 168,A 166.7358,B 10.6517,C 0.1185,E1 10.4968,E2 284.0935} C_DIS
LIN {X -130.3758,Y 28.6673,Z 168,A 168.7033,B 10.6516,C 0.1219,E1 10.4956,E2 282.1161} C_DIS
LIN {X -131.0986,Y 25.1511,Z 168,A 170.8091,B 10.6516,C 0.1155,E1 10.4944,E2 279.9438} C_DIS
LIN {X -131.9287,Y 20.3533,Z 168,A 172.3592,B 10.6514,C 0.132,E1 10.4938,E2 278.4612} C_DIS
LIN {X -132.5102,Y 16.143,Z 168,A 174.2034,B 10.6514,C 0.1369,E1 10.4931,E2 276.6166} C_DIS
LIN {X -132.8895,Y 12.6434,Z 168,A 175.7102,B 10.6514,C 0.1414,E1 10.4927,E2 275.1118} C_DIS
LIN {X -133.2005,Y 8.8008,Z 168,A 177.4592,B 10.6513,C 0.1445,E1 10.4923,E2 273.3532} C_DIS
LIN {X -133.398,Y 4.9526,Z 168,A 179.1291,B 10.6513,C 0.149,E1 10.4921,E2 271.6831} C_DIS
LIN {X -133.4904,Y 0.5007,Z 168,A -178.9885,B 10.6511,C 0.1551,E1 10.4921,E2 269.8062} C_DIS
LIN {X -133.453,Y -3.1726,Z 168,A -177.3578,B 10.6511,C 0.1587,E1 10.4921,E2 268.1704} C_DIS
LIN {X -133.3205,Y -6.7167,Z 168,A -175.8333,B 10.6511,C 0.1631,E1 10.4923,E2 266.6472} C_DIS
LIN {X -133.0457,Y -10.883,Z 168,A -174.0226,B 10.6509,C 0.168,E1 10.4927,E2 264.836} C_DIS
LIN {X -132.715,Y -14.359,Z 168,A -172.506,B 10.6509,C 0.172,E1 10.4931,E2 263.3187} C_DIS
LIN {X -132.2267,Y -18.3262,Z 168,A -170.7048,B 10.6509,C 0.1753,E1 10.4938,E2 261.5088} C_DIS
LIN {X -131.6917,Y -21.8348,Z 168,A -169.007,B 10.6509,C 0.1763,E1 10.4946,E2 259.7912} C_DIS
LIN {X -130.5018,Y -28.0837,Z 168,A -166.5619,B 10.6506,C 0.1896,E1 10.4959,E2 257.3832} C_DIS
LIN {X -129.8429,Y -30.989,Z 168,A -164.5641,B 10.6508,C 0.1793,E1 10.4972,E2 255.2991} C_DIS
LIN {X -128.6307,Y -35.6876,Z 168,A -163.0776,B 10.6505,C 0.1967,E1 10.4983,E2 253.887} C_DIS
LIN {X -127.3718,Y -39.9537,Z 168,A -161.0176,B 10.6505,C 0.1991,E1 10.4999,E2 251.8103} C_DIS
LIN {X -126.1699,Y -43.5953,Z 168,A -159.4976,B 10.6503,C 0.2061,E1 10.5013,E2 250.3069} C_DIS
LIN {X -125.0787,Y -46.634,Z 168,A -158.0231,B 10.6503,C 0.2081,E1 10.5027,E2 248.8227} C_DIS
LIN {X -123.6862,Y -50.2114,Z 168,A -156.3519,B 10.6502,C 0.2121,E1 10.5044,E2 247.1499} C_DIS
LIN {X -122.0959,Y -53.9656,Z 168,A -154.7171,B 10.65,C 0.219,E1 10.5062,E2 245.5305} C_DIS
LIN {X -120.6012,Y -57.2257,Z 168,A -152.772,B 10.6501,C 0.215,E1 10.5086,E2 243.5371} C_DIS
LIN {X -119.1879,Y -60.1151,Z 168,A -151.5757,B 10.65,C 0.2222,E1 10.5101,E2 242.3643} C_DIS
LIN {X -117.459,Y -63.4298,Z 168,A -150.0434,B 10.6499,C 0.2277,E1 10.5121,E2 240.8419} C_DIS
LIN {X -115.6188,Y -66.7248,Z 168,A -148.2975,B 10.6499,C 0.2292,E1 10.5145,E2 239.0817} C_DIS
LIN {X -113.3351,Y -70.5338,Z 168,A -146.3762,B 10.6497,C 0.2336,E1 10.5173,E2 237.1597} C_DIS
LIN {X -110.0042,Y -75.6239,Z 168,A -143.7673,B 10.6496,C 0.2399,E1 10.5213,E2 234.5526} C_DIS
LIN {X -107.409,Y -79.2671,Z 168,A -141.7656,B 10.6496,C 0.2426,E1 10.5246,E2 232.542} C_DIS
LIN {X -104.5464,Y -83.0057,Z 168,A -139.7364,B 10.6494,C 0.247,E1 10.5281,E2 230.5129} C_DIS
LIN {X -101.7016,Y -86.4677,Z 168,A -137.8193,B 10.6494,C 0.2513,E1 10.5315,E2 228.5974} C_DIS
LIN {X -98.8294,Y -89.7364,Z 168,A -135.936,B 10.6492,C 0.2549,E1 10.535,E2 226.713} C_DIS
LIN {X -95.8419,Y -92.9205,Z 168,A -134.0276,B 10.6492,C 0.2581,E1 10.5387,E2 224.8012} C_DIS
LIN {X -92.6196,Y -96.1332,Z 168,A -132.0397,B 10.6491,C 0.2612,E1 10.5427,E2 222.8097} C_DIS
LIN {X -89.3602,Y -99.1705,Z 168,A -130.1526,B 10.649,C 0.2653,E1 10.5466,E2 220.9264} C_DIS
LIN {X -84.7899,Y -103.1053,Z 168,A -127.5043,B 10.649,C 0.2688,E1 10.5522,E2 218.2716} C_DIS
LIN {X -81.4193,Y -105.7872,Z 168,A -125.6168,B 10.6488,C 0.2711,E1 10.5564,E2 216.3798} C_DIS
LIN {X -78.4827,Y -107.9832,Z 168,A -124.0311,B 10.6488,C 0.2734,E1 10.56,E2 214.7929} C_DIS
LIN {X -74.5818,Y -110.7137,Z 168,A -122.0185,B 10.6487,C 0.2773,E1 10.5646,E2 212.7846} C_DIS
LIN {X -70.4742,Y -113.3722,Z 168,A -119.6588,B 10.6487,C 0.2749,E1 10.5702,E2 210.3932} C_DIS
LIN {X -67.604,Y -115.1068,Z 168,A -118.484,B 10.6486,C 0.2825,E1 10.573,E2 209.2512} C_DIS
LIN {X -64.282,Y -116.9951,Z 168,A -117.0383,B 10.6484,C 0.2888,E1 10.5764,E2 207.8295} C_DIS
LIN {X -61.521,Y -118.4689,Z 168,A -115.4063,B 10.6485,C 0.2843,E1 10.5806,E2 206.1621} C_DIS
LIN {X -57.9316,Y -120.2641,Z 168,A -113.7681,B 10.6485,C 0.2881,E1 10.5846,E2 204.5343} C_DIS
LIN {X -54.6751,Y -121.7785,Z 168,A -112.4686,B 10.6482,C 0.295,E1 10.5879,E2 203.2645} C_DIS
LIN {X -50.8557,Y -123.4239,Z 168,A -110.325,B 10.6484,C 0.2892,E1 10.5935,E2 201.0767} C_DIS
LIN {X -47.1918,Y -124.8698,Z 168,A -108.717,B 10.6483,C 0.2925,E1 10.5977,E2 199.4788} C_DIS
LIN {X -41.9697,Y -126.72,Z 168,A -106.0233,B 10.6484,C 0.2876,E1 10.6049,E2 196.7458} C_DIS
LIN {X -38.6056,Y -127.7859,Z 168,A -104.7552,B 10.6482,C 0.2941,E1 10.6082,E2 195.5079} C_DIS
LIN {X -34.5442,Y -128.9423,Z 168,A -103.1072,B 10.6482,C 0.2989,E1 10.6126,E2 193.88} C_DIS
LIN {X -31.4322,Y -129.7361,Z 168,A -101.6281,B 10.6482,C 0.2975,E1 10.6166,E2 192.3881} C_DIS
LIN {X -27.9321,Y -130.5346,Z 168,A -100.0637,B 10.6482,C 0.2978,E1 10.6209,E2 190.8205} C_DIS
LIN {X -23.6944,Y -131.3698,Z 168,A -98.2389,B 10.6482,C 0.2992,E1 10.6259,E2 188.9988} C_DIS
LIN {X -20.2844,Y -131.9394,Z 168,A -96.7374,B 10.6481,C 0.2993,E1 10.63,E2 187.4946} C_DIS
LIN {X -16.1925,Y -132.5043,Z 168,A -94.9562,B 10.6481,C 0.2996,E1 10.635,E2 185.7118} C_DIS
LIN {X -12.8895,Y -132.8659,Z 168,A -93.5024,B 10.6481,C 0.2992,E1 10.639,E2 184.254} C_DIS
LIN {X -8.7496,Y -133.2037,Z 168,A -91.7109,B 10.6481,C 0.2992,E1 10.644,E2 182.4608} C_DIS
LIN {X -5.1247,Y -133.3913,Z 168,A -90.1848,B 10.6481,C 0.2999,E1 10.6483,E2 180.9379} C_DIS
LIN {X -1.0765,Y -133.4858,Z 168,A -88.4401,B 10.6481,C 0.2996,E1 10.6531,E2 179.1916} C_DIS
LIN {X -1.0765,Y -133.4858,Z 168,A -88.4401,B 10.6481,C 0.2996,E1 10.6531,E2 179.1916} C_DIS
Enddeposition()
LIN {X 0.9781,Y -134.3988,Z 168,A -87.5566,B 10.4281,C 0.3146,E1 10.4358,E2 178.4067} C_DIS
Startdeposition()
$VEL.CP = VEL_PRINT
LIN {X -3.0582,Y -134.3706,Z 168,A -89.9687,B 10.4276,C 0.3303,E1 10.4289,E2 180.9055} C_DIS
LIN {X -6.8549,Y -134.2287,Z 168,A -91.4986,B 10.4276,C 0.3283,E1 10.4246,E2 182.4249} C_DIS
LIN {X -11.3739,Y -133.9215,Z 168,A -93.411,B 10.4276,C 0.3277,E1 10.4193,E2 184.3358} C_DIS
LIN {X -15.0799,Y -133.5567,Z 168,A -95.1306,B 10.4276,C 0.3304,E1 10.4145,E2 186.0723} C_DIS
LIN {X -19.071,Y -133.0436,Z 168,A -96.7462,B 10.4276,C 0.3277,E1 10.41,E2 187.6761} C_DIS
LIN {X -23.0674,Y -132.4106,Z 168,A -98.5197,B 10.4276,C 0.3282,E1 10.4051,E2 189.4562} C_DIS
LIN {X -26.6964,Y -131.7254,Z 168,A -100.0262,B 10.4277,C 0.326,E1 10.401,E2 190.9548} C_DIS
LIN {X -30.1472,Y -130.9788,Z 168,A -101.5792,B 10.4277,C 0.3263,E1 10.3968,E2 192.514} C_DIS
LIN {X -34.3923,Y -129.9287,Z 168,A -103.4454,B 10.4277,C 0.3252,E1 10.3917,E2 194.3809} C_DIS
LIN {X -37.8699,Y -128.9578,Z 168,A -104.9486,B 10.4278,C 0.3234,E1 10.3877,E2 195.8799} C_DIS
LIN {X -42.6989,Y -127.4406,Z 168,A -107.1035,B 10.4278,C 0.3216,E1 10.382,E2 198.0347} C_DIS
LIN {X -46.4421,Y -126.1266,Z 168,A -108.7683,B 10.4279,C 0.3196,E1 10.3776,E2 199.6966} C_DIS
LIN {X -50.0001,Y -124.7569,Z 168,A -110.763,B 10.4278,C 0.3258,E1 10.3723,E2 201.7366} C_DIS
LIN {X -53.1246,Y -123.4586,Z 168,A -111.976,B 10.4279,C 0.3195,E1 10.3692,E2 202.9216} C_DIS
LIN {X -56.5925,Y -121.9078,Z 168,A -113.525,B 10.428,C 0.3163,E1 10.3653,E2 204.462} C_DIS
LIN {X -59.7185,Y -120.4075,Z 168,A -115.0306,B 10.428,C 0.3151,E1 10.3615,E2 205.9709} C_DIS
LIN {X -63.2126,Y -118.6129,Z 168,A -116.8256,B 10.428,C 0.3156,E1 10.3571,E2 207.7807} C_DIS
LIN {X -66.9075,Y -116.5686,Z 168,A -118.7234,B 10.428,C 0.3152,E1 10.3524,E2 209.6903} C_DIS
LIN {X -71.4412,Y -113.8464,Z 168,A -120.7198,B 10.4283,C 0.3067,E1 10.3477,E2 211.6549} C_DIS
LIN {X -74.3582,Y -111.9629,Z 168,A -122.3942,B 10.4283,C 0.3084,E1 10.3438,E2 213.3528} C_DIS
LIN {X -78.1061,Y -109.3809,Z 168,A -124.3236,B 10.4283,C 0.3051,E1 10.3394,E2 215.2805} C_DIS
LIN {X -80.9422,Y -107.299,Z 168,A -125.6161,B 10.4286,C 0.2984,E1 10.3365,E2 216.5473} C_DIS
LIN {X -83.5983,Y -105.2429,Z 168,A -127.4268,B 10.4284,C 0.3036,E1 10.3325,E2 218.404} C_DIS
LIN {X -88.3538,Y -101.2834,Z 168,A -129.9337,B 10.4286,C 0.2962,E1 10.3272,E2 220.8941} C_DIS
LIN {X -91.7988,Y -98.1722,Z 168,A -131.9305,B 10.4287,C 0.2929,E1 10.323,E2 222.8925} C_DIS
LIN {X -95.0485,Y -95.0299,Z 168,A -133.9131,B 10.4287,C 0.2902,E1 10.3191,E2 224.8812} C_DIS
LIN {X -98.1915,Y -91.778,Z 168,A -135.8493,B 10.4289,C 0.2864,E1 10.3154,E2 226.8175} C_DIS
LIN {X -101.1372,Y -88.5214,Z 168,A -137.7057,B 10.429,C 0.2821,E1 10.3119,E2 228.6712} C_DIS
LIN {X -103.8842,Y -85.2812,Z 168,A -139.5623,B 10.429,C 0.2791,E1 10.3086,E2 230.5325} C_DIS
LIN {X -106.5975,Y -81.8644,Z 168,A -141.4575,B 10.4292,C 0.2756,E1 10.3053,E2 232.4311} C_DIS
LIN {X -108.5225,Y -79.2951,Z 168,A -142.8414,B 10.4292,C 0.2728,E1 10.303,E2 233.8161} C_DIS
LIN {X -111.6445,Y -74.8346,Z 168,A -145.2085,B 10.4294,C 0.2682,E1 10.2993,E2 236.1875} C_DIS
LIN {X -113.8918,Y -71.3693,Z 168,A -146.9123,B 10.4295,C 0.2629,E1 10.2967,E2 237.8834} C_DIS
LIN {X -116.1183,Y -67.6863,Z 168,A -148.8429,B 10.4295,C 0.2602,E1 10.294,E2 239.8244} C_DIS
LIN {X -118.4409,Y -63.5334,Z 168,A -150.9249,B 10.4297,C 0.2562,E1 10.2912,E2 241.9115} C_DIS
LIN {X -120.7018,Y -59.122,Z 168,A -153.3217,B 10.4297,C 0.2562,E1 10.2881,E2 244.3411} C_DIS
LIN {X -122.4063,Y -55.5101,Z 168,A -154.5606,B 10.43,C 0.2428,E1 10.2868,E2 245.5228} C_DIS
LIN {X -124.1137,Y -51.5757,Z 168,A -156.4508,B 10.43,C 0.2392,E1 10.2847,E2 247.4191} C_DIS
LIN {X -125.4206,Y -48.3121,Z 168,A -158.1255,B 10.43,C 0.2385,E1 10.2829,E2 249.1139} C_DIS
LIN {X -126.96,Y -44.1067,Z 168,A -159.9741,B 10.4302,C 0.2321,E1 10.2812,E2 250.9538} C_DIS
LIN {X -128.2762,Y -40.126,Z 168,A -161.9241,B 10.4302,C 0.2303,E1 10.2795,E2 252.922} C_DIS
LIN {X -129.3553,Y -36.4902,Z 168,A -163.4995,B 10.4304,C 0.225,E1 10.2783,E2 254.491} C_DIS
LIN {X -130.9452,Y -30.2943,Z 168,A -165.9606,B 10.4306,C 0.2123,E1 10.2767,E2 256.9178} C_DIS
LIN {X -131.8221,Y -26.2212,Z 168,A -168.4034,B 10.4305,C 0.2198,E1 10.2753,E2 259.4392} C_DIS
LIN {X -132.5418,Y -22.293,Z 168,A -169.6517,B 10.4308,C 0.2064,E1 10.2747,E2 260.6315} C_DIS
LIN {X -133.0607,Y -18.9511,Z 168,A -171.1363,B 10.4308,C 0.2031,E1 10.2741,E2 262.1199} C_DIS
LIN {X -133.5493,Y -15.149,Z 168,A -172.9246,B 10.4308,C 0.2012,E1 10.2735,E2 263.9252} C_DIS
LIN {X -133.9377,Y -11.1817,Z 168,A -174.5839,B 10.431,C 0.1955,E1 10.2731,E2 265.578} C_DIS
LIN {X -134.2359,Y -6.7119,Z 168,A -176.501,B 10.431,C 0.1901,E1 10.2727,E2 267.4942} C_DIS
LIN {X -134.3821,Y -2.4156,Z 168,A -178.3468,B 10.4312,C 0.185,E1 10.2726,E2 269.3398} C_DIS
LIN {X -134.3872,Y 2.1104,Z 168,A 179.72,B 10.4312,C 0.1794,E1 10.2726,E2 271.2715} C_DIS
LIN {X -134.2988,Y 5.3093,Z 168,A 178.3407,B 10.4313,C 0.1757,E1 10.2728,E2 272.6512} C_DIS
LIN {X -134.0944,Y 9.1351,Z 168,A 176.5906,B 10.4313,C 0.1731,E1 10.2731,E2 274.4136} C_DIS
LIN {X -133.79,Y 12.8277,Z 168,A 175.0969,B 10.4315,C 0.1669,E1 10.2734,E2 275.8954} C_DIS
LIN {X -133.4127,Y 16.2939,Z 168,A 173.5165,B 10.4315,C 0.1643,E1 10.2739,E2 277.4855} C_DIS
LIN {X -132.2506,Y 23.9611,Z 168,A 170.3503,B 10.4317,C 0.1522,E1 10.2753,E2 280.6316} C_DIS
LIN {X -131.7195,Y 26.7254,Z 168,A 168.9878,B 10.4317,C 0.1517,E1 10.276,E2 282.0122} C_DIS
LIN {X -130.9967,Y 30.0689,Z 168,A 167.4791,B 10.4317,C 0.1485,E1 10.277,E2 283.5254} C_DIS
LIN {X -129.7726,Y 34.9777,Z 168,A 165.2619,B 10.4318,C 0.1435,E1 10.2785,E2 285.7474} C_DIS
LIN {X -128.5808,Y 39.1312,Z 168,A 163.4377,B 10.4318,C 0.1379,E1 10.2799,E2 287.5675} C_DIS
LIN {X -127.4959,Y 42.5328,Z 168,A 161.8858,B 10.4319,C 0.1342,E1 10.2813,E2 289.1214} C_DIS
LIN {X -126.3461,Y 45.836,Z 168,A 160.419,B 10.4319,C 0.1296,E1 10.2827,E2 290.5836} C_DIS
LIN {X -125.2204,Y 48.8271,Z 168,A 159.0168,B 10.432,C 0.1266,E1 10.2841,E2 291.9891} C_DIS
LIN {X -123.7378,Y 52.4758,Z 168,A 157.0376,B 10.432,C 0.1277,E1 10.2862,E2 294.0022} C_DIS
LIN {X -121.7856,Y 56.8569,Z 168,A 155.2933,B 10.4321,C 0.1165,E1 10.2882,E2 295.7085} C_DIS
LIN {X -119.8657,Y 60.7984,Z 168,A 153.6163,B 10.4322,C 0.108,E1 10.2902,E2 297.3605} C_DIS
LIN {X -118.6222,Y 63.1949,Z 168,A 152.1097,B 10.4322,C 0.1117,E1 10.2922,E2 298.9083} C_DIS
LIN {X -115.8475,Y 68.1476,Z 168,A 149.9134,B 10.4323,C 0.1012,E1 10.2952,E2 301.0753} C_DIS
LIN {X -112.709,Y 73.2216,Z 168,A 147.3363,B 10.4323,C 0.0955,E1 10.299,E2 303.6538} C_DIS
LIN {X -110.996,Y 75.7938,Z 168,A 145.7222,B 10.4323,C 0.0979,E1 10.3016,E2 305.3018} C_DIS
LIN {X -108.3605,Y 79.5156,Z 168,A 143.7804,B 10.4323,C 0.0932,E1 10.3048,E2 307.2412} C_DIS
LIN {X -105.5787,Y 83.174,Z 168,A 141.8058,B 10.4324,C 0.0888,E1 10.3081,E2 309.2155} C_DIS
LIN {X -102.7244,Y 86.675,Z 168,A 139.8574,B 10.4324,C 0.0849,E1 10.3116,E2 311.1646} C_DIS
LIN {X -99.8437,Y 89.9785,Z 168,A 137.9286,B 10.4324,C 0.0819,E1 10.3152,E2 313.0986} C_DIS
LIN {X -96.8001,Y 93.2447,Z 168,A 136.0028,B 10.4324,C 0.0782,E1 10.3189,E2 315.0251} C_DIS
LIN {X -93.6006,Y 96.4556,Z 168,A 134.0662,B 10.4325,C 0.0742,E1 10.3227,E2 316.9601} C_DIS
LIN {X -90.3434,Y 99.5128,Z 168,A 132.151,B 10.4325,C 0.0706,E1 10.3267,E2 318.8748} C_DIS
LIN {X -87.013,Y 102.4376,Z 168,A 130.2611,B 10.4325,C 0.0669,E1 10.3307,E2 320.7628} C_DIS
LIN {X -83.5122,Y 105.3115,Z 168,A 128.3102,B 10.4325,C 0.0637,E1 10.3349,E2 322.7142} C_DIS
LIN {X -80.0323,Y 107.9798,Z 168,A 126.3907,B 10.4326,C 0.0613,E1 10.3392,E2 324.6378} C_DIS
LIN {X -76.2933,Y 110.6533,Z 168,A 124.4548,B 10.4326,C 0.0575,E1 10.3436,E2 326.569} C_DIS
LIN {X -72.7393,Y 113.0214,Z 168,A 122.5743,B 10.4326,C 0.0557,E1 10.348,E2 328.455} C_DIS
LIN {X -68.8968,Y 115.4035,Z 168,A 120.6648,B 10.4326,C 0.0523,E1 10.3525,E2 330.3605} C_DIS
LIN {X -61.8889,Y 119.308,Z 168,A 117.3412,B 10.4326,C 0.0454,E1 10.3607,E2 333.6698} C_DIS
LIN {X -59.2897,Y 120.6191,Z 168,A 116.0556,B 10.4326,C 0.0447,E1 10.3639,E2 334.9595} C_DIS
LIN {X -56.22,Y 122.0801,Z 168,A 114.5891,B 10.4326,C 0.0431,E1 10.3676,E2 336.4269} C_DIS
LIN {X -51.527,Y 124.134,Z 168,A 112.3988,B 10.4327,C 0.0407,E1 10.3732,E2 338.6162} C_DIS
LIN {X -47.7379,Y 125.6412,Z 168,A 110.552,B 10.4327,C 0.041,E1 10.378,E2 340.4746} C_DIS
LIN {X -43.8549,Y 127.0473,Z 168,A 108.8405,B 10.4327,C 0.0382,E1 10.3825,E2 342.1788} C_DIS
LIN {X -38.1174,Y 128.8852,Z 168,A 105.9703,B 10.4327,C 0.042,E1 10.3903,E2 345.0828} C_DIS
LIN {X -34.8035,Y 129.8191,Z 168,A 104.8543,B 10.4327,C 0.0336,E1 10.3932,E2 346.1562} C_DIS
LIN {X -31.5561,Y 130.6464,Z 168,A 102.7793,B 10.4327,C 0.0459,E1 10.399,E2 348.3065} C_DIS
LIN {X -26.7295,Y 131.7187,Z 168,A 101.3424,B 10.4327,C 0.0306,E1 10.4027,E2 349.6629} C_DIS
LIN {X -23.6658,Y 132.3035,Z 168,A 99.9143,B 10.4327,C 0.0319,E1 10.4067,E2 351.1019} C_DIS
LIN {X -19.6496,Y 132.9609,Z 168,A 98.1197,B 10.4327,C 0.0324,E1 10.4116,E2 352.9025} C_DIS
LIN {X -15.9874,Y 133.4493,Z 168,A 96.6049,B 10.4327,C 0.0304,E1 10.4158,E2 354.4093} C_DIS
LIN {X -12.2687,Y 133.8437,Z 168,A 94.9417,B 10.4327,C 0.0314,E1 10.4204,E2 356.0798} C_DIS
LIN {X -8.2364,Y 134.151,Z 168,A 93.296,B 10.4327,C 0.0293,E1 10.425,E2 357.7152} C_DIS
LIN {X -4.3071,Y 134.3359,Z 168,A 91.5394,B 10.4327,C 0.0307,E1 10.4299,E2 359.4805} C_DIS
LIN {X -0.2709,Y 134.4043,Z 168,A 89.854,B 10.4327,C 0.0299,E1 10.4346,E2 361.1609} C_DIS
LIN {X 3.7509,Y 134.3513,Z 168,A 88.199,B 10.4327,C 0.0286,E1 10.4392,E2 362.808} C_DIS
LIN {X 7.3184,Y 134.2054,Z 168,A 86.5398,B 10.4327,C 0.0317,E1 10.4439,E2 364.4829} C_DIS
LIN {X 11.418,Y 133.9177,Z 168,A 84.937,B 10.4327,C 0.0288,E1 10.4483,E2 366.0672} C_DIS
LIN {X 14.6647,Y 133.6014,Z 168,A 83.4402,B 10.4327,C 0.0315,E1 10.4525,E2 367.5762} C_DIS
LIN {X 18.8157,Y 133.0801,Z 168,A 81.7372,B 10.4327,C 0.0303,E1 10.4572,E2 369.269} C_DIS
LIN {X 22.4067,Y 132.5229,Z 168,A 80.1309,B 10.4327,C 0.0323,E1 10.4616,E2 370.8818} C_DIS
LIN {X 26.6821,Y 131.7283,Z 168,A 78.3422,B 10.4327,C 0.0318,E1 10.4665,E2 372.6622} C_DIS
LIN {X 29.8929,Y 131.0369,Z 168,A 76.9298,B 10.4327,C 0.0329,E1 10.4704,E2 374.0757} C_DIS
LIN {X 33.2618,Y 130.2227,Z 168,A 75.4998,B 10.4327,C 0.0328,E1 10.4742,E2 375.4998} C_DIS
LIN {X 36.9218,Y 129.2346,Z 168,A 73.6511,B 10.4327,C 0.0392,E1 10.4793,E2 377.3759} C_DIS
LIN {X 41.3819,Y 127.875,Z 168,A 71.794,B 10.4327,C 0.0379,E1 10.4842,E2 379.2171} C_DIS
LIN {X 44.6618,Y 126.7675,Z 168,A 70.3086,B 10.4327,C 0.0395,E1 10.4881,E2 380.7036} C_DIS
LIN {X 49.7919,Y 124.8405,Z 168,A 68.0139,B 10.4327,C 0.0409,E1 10.4941,E2 382.9931} C_DIS
LIN {X 53.5667,Y 123.2675,Z 168,A 66.3658,B 10.4327,C 0.0407,E1 10.4983,E2 384.6298} C_DIS
LIN {X 56.8667,Y 121.781,Z 168,A 64.8425,B 10.4327,C 0.042,E1 10.5021,E2 386.1508} C_DIS
LIN {X 60.2361,Y 120.1519,Z 168,A 63.023,B 10.4327,C 0.0492,E1 10.5067,E2 387.9971} C_DIS
LIN {X 63.3469,Y 118.5411,Z 168,A 61.7025,B 10.4327,C 0.0472,E1 10.51,E2 389.2971} C_DIS
LIN {X 68.7146,Y 115.5121,Z 168,A 59.2096,B 10.4327,C 0.0478,E1 10.516,E2 391.7742} C_DIS
LIN {X 71.9829,Y 113.5045,Z 168,A 57.4706,B 10.4327,C 0.0527,E1 10.5201,E2 393.5259} C_DIS
LIN {X 75.4896,Y 111.2029,Z 168,A 55.0729,B 10.4326,C 0.0697,E1 10.5258,E2 395.9963} C_DIS
LIN {X 79.8768,Y 108.0951,Z 168,A 53.6508,B 10.4326,C 0.0532,E1 10.5288,E2 397.3153} C_DIS
LIN {X 84.5224,Y 104.5023,Z 168,A 51.084,B 10.4326,C 0.0592,E1 10.5345,E2 399.8904} C_DIS
LIN {X 87.3187,Y 102.1777,Z 168,A 49.3634,B 10.4326,C 0.0661,E1 10.5382,E2 401.632} C_DIS
LIN {X 90.6609,Y 99.2245,Z 168,A 47.4751,B 10.4326,C 0.0694,E1 10.5421,E2 403.5193} C_DIS
LIN {X 93.8855,Y 96.1787,Z 168,A 45.6246,B 10.4326,C 0.0722,E1 10.5458,E2 405.3657} C_DIS
LIN {X 96.8899,Y 93.1516,Z 168,A 43.7992,B 10.4326,C 0.0761,E1 10.5494,E2 407.1926} C_DIS
LIN {X 99.878,Y 89.9403,Z 168,A 41.9955,B 10.4325,C 0.0785,E1 10.5528,E2 408.9892} C_DIS
LIN {X 102.706,Y 86.697,Z 168,A 40.1209,B 10.4325,C 0.0835,E1 10.5562,E2 410.8694} C_DIS
LIN {X 107.025,Y 81.3054,Z 168,A 37.4631,B 10.4325,C 0.0832,E1 10.5608,E2 413.4941} C_DIS
LIN {X 108.839,Y 78.8594,Z 168,A 35.7373,B 10.4323,C 0.0966,E1 10.5637,E2 415.2721} C_DIS
LIN {X 110.79,Y 76.094,Z 168,A 34.7378,B 10.4324,C 0.0892,E1 10.5652,E2 416.2191} C_DIS
LIN {X 112.5565,Y 73.4566,Z 168,A 33.165,B 10.4324,C 0.0978,E1 10.5677,E2 417.8192} C_DIS
LIN {X 114.9905,Y 69.584,Z 168,A 30.6699,B 10.4321,C 0.1159,E1 10.5714,E2 420.3808} C_DIS
LIN {X 117.6943,Y 64.9063,Z 168,A 29.1668,B 10.4323,C 0.1022,E1 10.5733,E2 421.7893} C_DIS
LIN {X 119.4422,Y 61.6303,Z 168,A 27.2028,B 10.4322,C 0.1156,E1 10.5759,E2 423.8003} C_DIS
LIN {X 120.9673,Y 58.5799,Z 168,A 26.1417,B 10.4322,C 0.1097,E1 10.5772,E2 424.815} C_DIS
LIN {X 122.8465,Y 54.526,Z 168,A 24.1436,B 10.4322,C 0.117,E1 10.5795,E2 426.8258} C_DIS
LIN {X 124.5768,Y 50.4468,Z 168,A 21.9538,B 10.432,C 0.1295,E1 10.5819,E2 429.0533} C_DIS
LIN {X 125.95,Y 46.9135,Z 168,A 20.739,B 10.432,C 0.124,E1 10.583,E2 430.2209} C_DIS
LIN {X 127.3136,Y 43.0802,Z 168,A 18.2671,B 10.4318,C 0.147,E1 10.5853,E2 432.783} C_DIS
LIN {X 129.038,Y 37.5962,Z 168,A 16.5808,B 10.4319,C 0.1349,E1 10.5866,E2 434.3793} C_DIS
LIN {X 129.9318,Y 34.3808,Z 168,A 15.1948,B 10.4319,C 0.138,E1 10.5876,E2 435.762} C_DIS
LIN {X 130.9529,Y 30.2608,Z 168,A 13.3819,B 10.4319,C 0.1432,E1 10.5888,E2 437.5769} C_DIS
LIN {X 131.712,Y 26.7621,Z 168,A 11.9469,B 10.4318,C 0.1452,E1 10.5896,E2 439.0022} C_DIS
LIN {X 132.3286,Y 23.5252,Z 168,A 10.5265,B 10.4318,C 0.1497,E1 10.5903,E2 440.4257} C_DIS
LIN {X 133.0003,Y 19.3741,Z 168,A 8.7244,B 10.4316,C 0.1551,E1 10.5911,E2 442.2307} C_DIS
LIN {X 133.4813,Y 15.7187,Z 168,A 7.2526,B 10.4316,C 0.1571,E1 10.5916,E2 443.6918} C_DIS
LIN {X 133.8636,Y 12.0587,Z 168,A 5.5441,B 10.4315,C 0.1652,E1 10.5921,E2 445.4188} C_DIS
LIN {X 134.1534,Y 8.1975,Z 168,A 4.0391,B 10.4315,C 0.1663,E1 10.5924,E2 446.9076} C_DIS
LIN {X 134.3411,Y 4.1187,Z 168,A 2.2799,B 10.4314,C 0.1719,E1 10.5925,E2 448.6708} C_DIS
LIN {X 134.4078,Y -0.0206,Z 168,A 0.4152,B 10.4313,C 0.1796,E1 10.5925,E2 450.5496} C_DIS
LIN {X 134.3398,Y -4.1641,Z 168,A -1.1239,B 10.4313,C 0.179,E1 10.5925,E2 452.0626} C_DIS
LIN {X 134.2202,Y -7.0252,Z 168,A -2.7612,B 10.431,C 0.1931,E1 10.5922,E2 453.7519} C_DIS
LIN {X 133.9589,Y -10.9311,Z 168,A -3.8192,B 10.4312,C 0.1826,E1 10.592,E2 454.7371} C_DIS
LIN {X 133.6484,Y -14.2277,Z 168,A -5.3987,B 10.4311,C 0.191,E1 10.5916,E2 456.3387} C_DIS
LIN {X 133.2188,Y -17.809,Z 168,A -7.0313,B 10.4309,C 0.1979,E1 10.591,E2 457.9845} C_DIS
LIN {X 132.5854,Y -22.0321,Z 168,A -8.7077,B 10.4309,C 0.1995,E1 10.5903,E2 459.6452} C_DIS
LIN {X 131.9862,Y -25.376,Z 168,A -10.1251,B 10.4309,C 0.2029,E1 10.5896,E2 461.0604} C_DIS
LIN {X 131.2067,Y -29.1495,Z 168,A -11.864,B 10.4307,C 0.2101,E1 10.5885,E2 462.813} C_DIS
LIN {X 129.2537,Y -36.8537,Z 168,A -15.0597,B 10.4306,C 0.215,E1 10.5863,E2 465.9887} C_DIS
LIN {X 128.2628,Y -40.168,Z 168,A -16.7639,B 10.4304,C 0.2249,E1 10.5849,E2 467.7228} C_DIS
LIN {X 126.7473,Y -44.7201,Z 168,A -18.5037,B 10.4304,C 0.223,E1 10.5833,E2 469.4274} C_DIS
LIN {X 125.598,Y -47.8532,Z 168,A -20.0541,B 10.4303,C 0.2301,E1 10.5818,E2 470.995} C_DIS
LIN {X 124.5338,Y -50.5535,Z 168,A -21.2044,B 10.4303,C 0.2314,E1 10.5806,E2 472.136} C_DIS
LIN {X 122.8694,Y -54.4747,Z 168,A -23.4033,B 10.4299,C 0.2459,E1 10.5781,E2 474.3838} C_DIS
LIN {X 121.2166,Y -58.0581,Z 168,A -24.6771,B 10.4301,C 0.2402,E1 10.5766,E2 475.6095} C_DIS
LIN {X 119.4562,Y -61.6027,Z 168,A -26.4179,B 10.4299,C 0.2461,E1 10.5744,E2 477.3587} C_DIS
LIN {X 117.3001,Y -65.6162,Z 168,A -28.3089,B 10.4299,C 0.2499,E1 10.5719,E2 479.2456} C_DIS
LIN {X 115.3452,Y -68.9946,Z 168,A -29.9398,B 10.4297,C 0.2533,E1 10.5696,E2 480.8744} C_DIS
LIN {X 113.0214,Y -72.7393,Z 168,A -31.7532,B 10.4297,C 0.2565,E1 10.5669,E2 482.6818} C_DIS
LIN {X 110.6228,Y -76.3377,Z 168,A -33.6334,B 10.4295,C 0.262,E1 10.564,E2 484.5685} C_DIS
LIN {X 108.0795,Y -79.8982,Z 168,A -35.4505,B 10.4295,C 0.2653,E1 10.561,E2 486.3817} C_DIS
LIN {X 105.4527,Y -83.3344,Z 168,A -37.3795,B 10.4293,C 0.2718,E1 10.5576,E2 488.3231} C_DIS
LIN {X 101.3529,Y -88.2742,Z 168,A -39.8741,B 10.4293,C 0.2722,E1 10.5532,E2 490.7909} C_DIS
LIN {X 98.4804,Y -91.4678,Z 168,A -41.6511,B 10.4293,C 0.275,E1 10.5499,E2 492.5632} C_DIS
LIN {X 93.0401,Y -96.9965,Z 168,A -45.9173,B 10.4284,C 0.3054,E1 10.5412,E2 496.9504} C_DIS
LIN {X 88.147,Y -101.4638,Z 168,A -48.6536,B 10.4283,C 0.309,E1 10.5354,E2 499.6789} C_DIS
LIN {X 83.2948,Y -105.4837,Z 168,A -50.2815,B 10.4288,C 0.2886,E1 10.5322,E2 501.1797} C_DIS
LIN {X 79.7202,Y -108.2102,Z 168,A -52.2715,B 10.4287,C 0.294,E1 10.5277,E2 503.1807} C_DIS
LIN {X 76.9218,Y -110.217,Z 168,A -54.247,B 10.4283,C 0.3088,E1 10.523,E2 505.2201} C_DIS
LIN {X 73.5944,Y -112.4654,Z 168,A -55.5988,B 10.4284,C 0.3031,E1 10.52,E2 506.5292} C_DIS
LIN {X 69.8301,Y -114.8416,Z 168,A -57.4631,B 10.4284,C 0.3054,E1 10.5156,E2 508.3912} C_DIS
LIN {X 66.0828,Y -117.0379,Z 168,A -59.3414,B 10.4283,C 0.309,E1 10.511,E2 510.2745} C_DIS
LIN {X 62.1612,Y -119.165,Z 168,A -61.1452,B 10.4283,C 0.3095,E1 10.5066,E2 512.0678} C_DIS
LIN {X 58.4204,Y -121.0435,Z 168,A -62.9695,B 10.4281,C 0.3129,E1 10.502,E2 513.8986} C_DIS
LIN {X 54.9515,Y -122.6562,Z 168,A -64.525,B 10.4281,C 0.3133,E1 10.4981,E2 515.4462} C_DIS
LIN {X 51.6872,Y -124.0671,Z 168,A -66.0727,B 10.4281,C 0.3159,E1 10.4941,E2 516.9991} C_DIS
LIN {X 48.0542,Y -125.5209,Z 168,A -67.6303,B 10.4281,C 0.3153,E1 10.4901,E2 518.5444} C_DIS
LIN {X 45.5429,Y -126.4518,Z 168,A -69.116,B 10.4278,C 0.3247,E1 10.4861,E2 520.0734} C_DIS
LIN {X 42.363,Y -127.5524,Z 168,A -70.6816,B 10.4276,C 0.3292,E1 10.4819,E2 521.6561} C_DIS
LIN {X 38.3699,Y -128.8115,Z 168,A -71.9225,B 10.428,C 0.3183,E1 10.4787,E2 522.8316} C_DIS
LIN {X 32.6959,Y -130.3663,Z 168,A -74.4793,B 10.4279,C 0.3217,E1 10.4718,E2 525.3962} C_DIS
LIN {X 29.6881,Y -131.0837,Z 168,A -75.8123,B 10.4279,C 0.323,E1 10.4682,E2 526.732} C_DIS
LIN {X 26.5346,Y -131.7583,Z 168,A -77.1553,B 10.4279,C 0.3233,E1 10.4645,E2 528.0719} C_DIS
LIN {X 23.5175,Y -132.33,Z 168,A -78.4983,B 10.4278,C 0.3249,E1 10.4608,E2 529.42} C_DIS
LIN {X 19.3741,Y -133.0003,Z 168,A -80.3267,B 10.4278,C 0.3269,E1 10.4557,E2 531.2544} C_DIS
LIN {X 15.7187,Y -133.4813,Z 168,A -81.8583,B 10.4278,C 0.3267,E1 10.4515,E2 532.7819} C_DIS
LIN {X 11.5833,Y -133.9038,Z 168,A -83.6384,B 10.4277,C 0.3276,E1 10.4465,E2 534.5641} C_DIS
LIN {X 8.2426,Y -134.1506,Z 168,A -85.0269,B 10.4277,C 0.3272,E1 10.4427,E2 535.9484} C_DIS
LIN {X 4.9544,Y -134.3126,Z 168,A -86.5443,B 10.4277,C 0.3301,E1 10.4384,E2 537.4807} C_DIS
LIN {X 0.9781,Y -134.3988,Z 168,A -87.5545,B 10.4281,C 0.315,E1 10.4358,E2 538.4067} C_DIS
Enddeposition()
LIN {X 0.9781,Y -134.3988,Z 168,A -87.5545,B 10.4281,C 0.315,E1 10.4358,E2 538.4067} C_DIS
Startdeposition()
$VEL.CP = VEL_PRINT
LIN {X 3.2328,Y -135.2801,Z 168,A -86.4717,B 10.3673,C 0.3204,E1 10.3782,E2 537.3597} C_DIS
LIN {X 6.624,Y -135.1555,Z 168,A -85.0208,B 10.3673,C 0.3197,E1 10.3822,E2 535.9062} C_DIS
LIN {X 10.6313,Y -134.9014,Z 168,A -83.2494,B 10.3673,C 0.3175,E1 10.3871,E2 534.125} C_DIS
LIN {X 14.6908,Y -134.5179,Z 168,A -81.5363,B 10.3673,C 0.3171,E1 10.3919,E2 532.4126} C_DIS
LIN {X 18.4583,Y -134.0544,Z 168,A -79.9175,B 10.3674,C 0.316,E1 10.3964,E2 530.7914} C_DIS
LIN {X 22.2277,Y -133.4794,Z 168,A -78.3993,B 10.3674,C 0.3173,E1 10.4006,E2 529.2842} C_DIS
LIN {X 26.2449,Y -132.75,Z 168,A -76.5142,B 10.3675,C 0.3125,E1 10.4058,E2 527.3783} C_DIS
LIN {X 30.3888,Y -131.8612,Z 168,A -74.8776,B 10.3675,C 0.3148,E1 10.4102,E2 525.7603} C_DIS
LIN {X 35.2111,Y -130.6563,Z 168,A -72.7923,B 10.3675,C 0.3135,E1 10.4158,E2 523.676} C_DIS
LIN {X 38.2342,Y -129.8035,Z 168,A -70.3277,B 10.3683,C 0.2852,E1 10.4229,E2 521.0659} C_DIS
LIN {X 45.7515,Y -127.3482,Z 168,A -67.664,B 10.3679,C 0.298,E1 10.4296,E2 518.4874} C_DIS
LIN {X 49.9167,Y -125.7759,Z 168,A -66.21,B 10.3677,C 0.3061,E1 10.4332,E2 517.0866} C_DIS
LIN {X 53.6434,Y -124.2301,Z 168,A -64.6297,B 10.3677,C 0.307,E1 10.4373,E2 515.5209} C_DIS
LIN {X 56.6243,Y -122.9001,Z 168,A -63.2092,B 10.3677,C 0.3043,E1 10.4409,E2 514.0944} C_DIS
LIN {X 59.7169,Y -121.4275,Z 168,A -61.8995,B 10.3677,C 0.3057,E1 10.4441,E2 512.8012} C_DIS
LIN {X 62.6593,Y -119.9358,Z 168,A -60.3689,B 10.3679,C 0.3004,E1 10.448,E2 511.2526} C_DIS
LIN {X 66.551,Y -117.8232,Z 168,A -58.4188,B 10.368,C 0.2957,E1 10.4528,E2 509.2913} C_DIS
LIN {X 69.9509,Y -115.8367,Z 168,A -56.4772,B 10.3683,C 0.2864,E1 10.4575,E2 507.3134} C_DIS
LIN {X 73.1954,Y -113.8146,Z 168,A -54.5178,B 10.3686,C 0.2752,E1 10.4622,E2 505.3091} C_DIS
LIN {X 77.917,Y -110.6354,Z 168,A -52.9901,B 10.3681,C 0.2927,E1 10.4655,E2 503.891} C_DIS
LIN {X 82.0721,Y -107.5893,Z 168,A -50.5653,B 10.3684,C 0.2827,E1 10.471,E2 501.4335} C_DIS
LIN {X 85.9238,Y -104.5394,Z 168,A -48.5317,B 10.3684,C 0.2798,E1 10.4754,E2 499.4038} C_DIS
LIN {X 89.2809,Y -101.6874,Z 168,A -46.3957,B 10.3687,C 0.2694,E1 10.48,E2 497.2316} C_DIS
LIN {X 92.143,Y -99.1006,Z 168,A -44.9385,B 10.3687,C 0.2704,E1 10.4829,E2 495.7949} C_DIS
LIN {X 95.9247,Y -95.4448,Z 168,A -42.9032,B 10.3687,C 0.2704,E1 10.4869,E2 493.7816} C_DIS
LIN {X 98.7018,Y -92.5708,Z 168,A -41.1929,B 10.3687,C 0.2662,E1 10.4902,E2 492.0672} C_DIS
LIN {X 101.6687,Y -89.3023,Z 168,A -39.539,B 10.3687,C 0.2674,E1 10.4932,E2 490.4384} C_DIS
LIN {X 105.9479,Y -84.1802,Z 168,A -36.6044,B 10.369,C 0.2581,E1 10.4985,E2 487.4872} C_DIS
LIN {X 108.6683,Y -80.6381,Z 168,A -34.7146,B 10.3691,C 0.2536,E1 10.5017,E2 485.5956} C_DIS
LIN {X 111.159,Y -77.1683,Z 168,A -32.9457,B 10.3691,C 0.2501,E1 10.5045,E2 483.8297} C_DIS
LIN {X 113.6743,Y -73.4133,Z 168,A -31.023,B 10.3693,C 0.2451,E1 10.5075,E2 481.9037} C_DIS
LIN {X 115.996,Y -69.6874,Z 168,A -29.1809,B 10.3694,C 0.2408,E1 10.5101,E2 480.0617} C_DIS
LIN {X 118.1139,Y -66.0337,Z 168,A -27.4228,B 10.3694,C 0.2369,E1 10.5126,E2 478.3054} C_DIS
LIN {X 120.0161,Y -62.5065,Z 168,A -25.8309,B 10.3695,C 0.2351,E1 10.5146,E2 476.7247} C_DIS
LIN {X 121.8236,Y -58.9077,Z 168,A -24.2368,B 10.3695,C 0.2333,E1 10.5166,E2 475.1428} C_DIS
LIN {X 122.9937,Y -56.4219,Z 168,A -22.8811,B 10.3698,C 0.2253,E1 10.5182,E2 473.7615} C_DIS
LIN {X 124.7106,Y -52.5181,Z 168,A -21.2011,B 10.3698,C 0.2236,E1 10.5201,E2 472.0953} C_DIS
LIN {X 127.1189,Y -46.3875,Z 168,A -18.6007,B 10.3698,C 0.2207,E1 10.5227,E2 469.5156} C_DIS
LIN {X 128.3633,Y -42.8208,Z 168,A -16.8689,B 10.37,C 0.2128,E1 10.5242,E2 467.7654} C_DIS
LIN {X 129.6592,Y -38.7271,Z 168,A -14.9859,B 10.3702,C 0.206,E1 10.5258,E2 465.8724} C_DIS
LIN {X 130.5611,Y -35.5682,Z 168,A -13.4239,B 10.3703,C 0.1977,E1 10.527,E2 464.2874} C_DIS
LIN {X 131.4016,Y -32.3234,Z 168,A -12.2642,B 10.3703,C 0.2003,E1 10.5277,E2 463.1588} C_DIS
LIN {X 132.1817,Y -28.965,Z 168,A -10.8728,B 10.3703,C 0.1978,E1 10.5286,E2 461.7743} C_DIS
LIN {X 132.8497,Y -25.7265,Z 168,A -9.4931,B 10.3703,C 0.1943,E1 10.5293,E2 460.3956} C_DIS
LIN {X 133.5086,Y -22.0522,Z 168,A -7.9456,B 10.3704,C 0.1905,E1 10.53,E2 458.8506} C_DIS
LIN {X 134.1254,Y -17.9252,Z 168,A -6.1832,B 10.3705,C 0.1855,E1 10.5307,E2 457.0869} C_DIS
LIN {X 134.5487,Y -14.404,Z 168,A -4.7106,B 10.3705,C 0.1819,E1 10.5312,E2 455.6164} C_DIS
LIN {X 134.9308,Y -10.224,Z 168,A -2.7157,B 10.3708,C 0.1711,E1 10.5317,E2 453.5924} C_DIS
LIN {X 135.2736,Y -3.4663,Z 168,A -0.0474,B 10.3708,C 0.1677,E1 10.532,E2 450.9458} C_DIS
LIN {X 135.3185,Y 0.4956,Z 168,A 1.631,B 10.3709,C 0.1628,E1 10.532,E2 449.2657} C_DIS
LIN {X 135.2216,Y 5.0999,Z 168,A 3.3841,B 10.3709,C 0.1621,E1 10.5318,E2 447.5352} C_DIS
LIN {X 135.0436,Y 8.611,Z 168,A 4.9462,B 10.371,C 0.1559,E1 10.5316,E2 445.9625} C_DIS
LIN {X 134.7079,Y 12.8313,Z 168,A 6.6629,B 10.371,C 0.1526,E1 10.5312,E2 444.2535} C_DIS
LIN {X 134.3167,Y 16.4321,Z 168,A 8.1987,B 10.3711,C 0.1481,E1 10.5307,E2 442.716} C_DIS
LIN {X 133.8017,Y 20.2031,Z 168,A 9.8099,B 10.3711,C 0.1435,E1 10.53,E2 441.1034} C_DIS
LIN {X 133.2189,Y 23.7391,Z 168,A 11.2145,B 10.3712,C 0.142,E1 10.5294,E2 439.7113} C_DIS
LIN {X 132.6242,Y 26.8629,Z 168,A 12.5607,B 10.3712,C 0.1381,E1 10.5286,E2 438.364} C_DIS
LIN {X 131.9025,Y 30.2079,Z 168,A 14.025,B 10.3713,C 0.1336,E1 10.5277,E2 436.8965} C_DIS
LIN {X 130.9391,Y 34.1506,Z 168,A 15.7834,B 10.3713,C 0.1278,E1 10.5265,E2 435.1318} C_DIS
LIN {X 129.9168,Y 37.8474,Z 168,A 17.7543,B 10.3716,C 0.1144,E1 10.525,E2 433.1163} C_DIS
LIN {X 128.6569,Y 41.9381,Z 168,A 19.2281,B 10.3716,C 0.118,E1 10.5238,E2 431.6832} C_DIS
LIN {X 127.327,Y 45.8102,Z 168,A 21.2344,B 10.3716,C 0.1064,E1 10.5218,E2 429.6416} C_DIS
LIN {X 125.8582,Y 49.7089,Z 168,A 22.6631,B 10.3716,C 0.1101,E1 10.5204,E2 428.2534} C_DIS
LIN {X 124.5077,Y 53.0014,Z 168,A 24.1511,B 10.3716,C 0.1065,E1 10.5188,E2 426.7665} C_DIS
LIN {X 122.974,Y 56.4646,Z 168,A 25.6447,B 10.3716,C 0.1051,E1 10.5171,E2 425.2854} C_DIS
LIN {X 121.0146,Y 60.5534,Z 168,A 27.6197,B 10.3717,C 0.0987,E1 10.5147,E2 423.3023} C_DIS
LIN {X 119.1489,Y 64.1468,Z 168,A 29.2641,B 10.3717,C 0.0961,E1 10.5125,E2 421.6654} C_DIS
LIN {X 117.5525,Y 67.0273,Z 168,A 30.7854,B 10.3717,C 0.0894,E1 10.5104,E2 420.1275} C_DIS
LIN {X 115.0322,Y 71.2665,Z 168,A 32.7586,B 10.3718,C 0.0871,E1 10.5076,E2 418.1673} C_DIS
LIN {X 112.5359,Y 75.146,Z 168,A 34.4634,B 10.3718,C 0.0885,E1 10.505,E2 416.492} C_DIS
LIN {X 110.633,Y 77.9204,Z 168,A 36.0744,B 10.3718,C 0.0805,E1 10.5024,E2 414.8572} C_DIS
LIN {X 107.9858,Y 81.5495,Z 168,A 37.8264,B 10.3718,C 0.0798,E1 10.4995,E2 413.1227} C_DIS
LIN {X 105.3855,Y 84.8832,Z 168,A 39.7392,B 10.3719,C 0.0728,E1 10.4962,E2 411.194} C_DIS
LIN {X 102.3408,Y 88.5308,Z 168,A 41.6662,B 10.3719,C 0.0704,E1 10.4927,E2 409.2765} C_DIS
LIN {X 99.4338,Y 91.7837,Z 168,A 43.5468,B 10.3719,C 0.0657,E1 10.4892,E2 407.391} C_DIS
LIN {X 96.3409,Y 95.0254,Z 168,A 45.4463,B 10.3719,C 0.0617,E1 10.4855,E2 405.4904} C_DIS
LIN {X 93.1391,Y 98.1657,Z 168,A 47.3243,B 10.372,C 0.0585,E1 10.4817,E2 403.6143} C_DIS
LIN {X 89.8167,Y 101.214,Z 168,A 49.2181,B 10.372,C 0.0552,E1 10.4778,E2 401.7217} C_DIS
LIN {X 86.24,Y 104.2781,Z 168,A 51.0377,B 10.372,C 0.0557,E1 10.4739,E2 399.923} C_DIS
LIN {X 82.9283,Y 106.9306,Z 168,A 52.9557,B 10.372,C 0.0496,E1 10.4697,E2 397.9897} C_DIS
LIN {X 79.3761,Y 109.5933,Z 168,A 54.9611,B 10.372,C 0.0434,E1 10.4651,E2 395.9685} C_DIS
LIN {X 74.9009,Y 112.6995,Z 168,A 57.0842,B 10.372,C 0.0441,E1 10.4603,E2 393.8675} C_DIS
LIN {X 71.2167,Y 115.0632,Z 168,A 58.8441,B 10.372,C 0.0435,E1 10.4562,E2 392.1188} C_DIS
LIN {X 66.6744,Y 117.7538,Z 168,A 61.2012,B 10.3721,C 0.0374,E1 10.4504,E2 389.7466} C_DIS
LIN {X 63.2946,Y 119.6022,Z 168,A 62.883,B 10.3721,C 0.034,E1 10.4463,E2 388.0584} C_DIS
LIN {X 59.035,Y 121.7629,Z 168,A 64.7814,B 10.3721,C 0.0344,E1 10.4416,E2 386.1751} C_DIS
LIN {X 55.4916,Y 123.4159,Z 168,A 66.3368,B 10.3721,C 0.0347,E1 10.4377,E2 384.6319} C_DIS
LIN {X 52.2932,Y 124.8045,Z 168,A 68.3646,B 10.3721,C 0.0203,E1 10.4323,E2 382.5367} C_DIS
LIN {X 47.9246,Y 126.5473,Z 168,A 69.8112,B 10.3721,C 0.0309,E1 10.4287,E2 381.157} C_DIS
LIN {X 45.058,Y 127.5975,Z 168,A 71.2315,B 10.3721,C 0.0268,E1 10.4249,E2 379.7213} C_DIS
LIN {X 41.217,Y 128.8872,Z 168,A 72.7436,B 10.3721,C 0.0299,E1 10.4209,E2 378.2342} C_DIS
LIN {X 37.8042,Y 129.9294,Z 168,A 74.3195,B 10.3721,C 0.0273,E1 10.4167,E2 376.6506} C_DIS
LIN {X 33.7847,Y 131.033,Z 168,A 76.1103,B 10.3721,C 0.0254,E1 10.4119,E2 374.857} C_DIS
LIN {X 30.2106,Y 131.9019,Z 168,A 77.6129,B 10.3721,C 0.0257,E1 10.4078,E2 373.3613} C_DIS
LIN {X 26.7472,Y 132.6478,Z 168,A 79.1256,B 10.3721,C 0.0246,E1 10.4037,E2 371.8476} C_DIS
LIN {X 22.8815,Y 133.3703,Z 168,A 80.8333,B 10.3721,C 0.0228,E1 10.3989,E2 370.1352} C_DIS
LIN {X 19.2308,Y 133.944,Z 168,A 82.3476,B 10.3721,C 0.0233,E1 10.3948,E2 368.6274} C_DIS
LIN {X 15.3125,Y 134.4503,Z 168,A 84.1172,B 10.3721,C 0.0207,E1 10.3898,E2 366.8467} C_DIS
LIN {X 11.4553,Y 134.8318,Z 168,A 85.6635,B 10.3721,C 0.0224,E1 10.3856,E2 365.3125} C_DIS
LIN {X 7.2462,Y 135.1242,Z 168,A 87.4726,B 10.3721,C 0.0217,E1 10.3805,E2 363.5014} C_DIS
LIN {X 3.3874,Y 135.2758,Z 168,A 89.1776,B 10.3721,C 0.02,E1 10.3757,E2 361.7886} C_DIS
LIN {X -0.7471,Y 135.3156,Z 168,A 90.8335,B 10.3721,C 0.0222,E1 10.3712,E2 360.145} C_DIS
LIN {X -4.891,Y 135.2298,Z 168,A 92.5731,B 10.3721,C 0.0227,E1 10.3663,E2 358.4082} C_DIS
LIN {X -8.3946,Y 135.057,Z 168,A 94.0799,B 10.3721,C 0.0225,E1 10.3621,E2 356.8994} C_DIS
LIN {X -12.5681,Y 134.7331,Z 168,A 95.858,B 10.3721,C 0.0229,E1 10.3572,E2 355.1217} C_DIS
LIN {X -15.6564,Y 134.4092,Z 168,A 97.015,B 10.3721,C 0.0268,E1 10.354,E2 353.9845} C_DIS
LIN {X -18.9693,Y 133.9814,Z 168,A 98.5715,B 10.3721,C 0.0244,E1 10.3496,E2 352.4116} C_DIS
LIN {X -22.1095,Y 133.4991,Z 168,A 99.9063,B 10.3721,C 0.0253,E1 10.346,E2 351.0789} C_DIS
LIN {X -25.5179,Y 132.8896,Z 168,A 101.22,B 10.3721,C 0.0293,E1 10.3424,E2 349.7846} C_DIS
LIN {X -28.8811,Y 132.1998,Z 168,A 102.9216,B 10.3721,C 0.025,E1 10.3377,E2 348.054} C_DIS
LIN {X -33.3039,Y 131.155,Z 168,A 104.7359,B 10.3721,C 0.0288,E1 10.3328,E2 346.2542} C_DIS
LIN {X -41.3,Y 128.8607,Z 168,A 107.9309,B 10.3721,C 0.0387,E1 10.3244,E2 343.1015} C_DIS
LIN {X -45.3225,Y 127.5029,Z 168,A 110.1827,B 10.3721,C 0.031,E1 10.3183,E2 340.7964} C_DIS
LIN {X -48.7984,Y 126.2122,Z 168,A 111.6815,B 10.3721,C 0.0342,E1 10.3144,E2 339.3074} C_DIS
LIN {X -52.297,Y 124.803,Z 168,A 113.2239,B 10.3721,C 0.0371,E1 10.3104,E2 337.7729} C_DIS
LIN {X -54.728,Y 123.7574,Z 168,A 114.4463,B 10.3721,C 0.0364,E1 10.3072,E2 336.5391} C_DIS
LIN {X -57.501,Y 122.4945,Z 168,A 115.8602,B 10.3721,C 0.0355,E1 10.3036,E2 335.1113} C_DIS
LIN {X -60.8864,Y 120.8465,Z 168,A 117.4138,B 10.3721,C 0.0385,E1 10.2998,E2 333.564} C_DIS
LIN {X -63.6219,Y 119.4303,Z 168,A 118.898,B 10.3721,C 0.0367,E1 10.2961,E2 332.0592} C_DIS
LIN {X -68.1134,Y 116.9271,Z 168,A 120.9285,B 10.3721,C 0.0429,E1 10.2912,E2 330.0484} C_DIS
LIN {X -71.8734,Y 114.6544,Z 168,A 122.7968,B 10.3721,C 0.0457,E1 10.2867,E2 328.1809} C_DIS
LIN {X -75.3901,Y 112.373,Z 168,A 124.5947,B 10.3721,C 0.0481,E1 10.2825,E2 326.3819} C_DIS
LIN {X -79.059,Y 109.8231,Z 168,A 126.5436,B 10.3721,C 0.0502,E1 10.2781,E2 324.4278} C_DIS
LIN {X -82.7047,Y 107.1039,Z 168,A 128.4625,B 10.3721,C 0.0539,E1 10.2738,E2 322.5116} C_DIS
LIN {X -86.2292,Y 104.287,Z 168,A 130.371,B 10.3721,C 0.0575,E1 10.2697,E2 320.6052} C_DIS
LIN {X -89.7331,Y 101.2879,Z 168,A 132.3403,B 10.372,C 0.061,E1 10.2656,E2 318.6359} C_DIS
LIN {X -92.9438,Y 98.3499,Z 168,A 134.1807,B 10.372,C 0.0648,E1 10.2618,E2 316.7977} C_DIS
LIN {X -95.9911,Y 95.378,Z 168,A 135.9981,B 10.372,C 0.0683,E1 10.2582,E2 314.9802} C_DIS
LIN {X -99.033,Y 92.2156,Z 168,A 137.8853,B 10.372,C 0.0717,E1 10.2546,E2 313.0914} C_DIS
LIN {X -102.0552,Y 88.8595,Z 168,A 139.8296,B 10.372,C 0.0753,E1 10.251,E2 311.1452} C_DIS
LIN {X -105.0018,Y 85.358,Z 168,A 141.8232,B 10.3719,C 0.0787,E1 10.2474,E2 309.1469} C_DIS
LIN {X -107.7613,Y 81.847,Z 168,A 143.7477,B 10.3719,C 0.0825,E1 10.2441,E2 307.2204} C_DIS
LIN {X -110.4324,Y 78.2048,Z 168,A 145.6391,B 10.3719,C 0.0875,E1 10.241,E2 305.3335} C_DIS
LIN {X -112.8747,Y 74.6367,Z 168,A 147.3389,B 10.3717,C 0.0945,E1 10.2384,E2 303.6516} C_DIS
LIN {X -115.2371,Y 70.9345,Z 168,A 149.5195,B 10.3717,C 0.093,E1 10.2351,E2 301.434} C_DIS
LIN {X -119.6291,Y 63.2434,Z 168,A 153.5237,B 10.3717,C 0.0978,E1 10.2297,E2 297.403} C_DIS
LIN {X -121.4284,Y 59.7149,Z 168,A 154.8322,B 10.3717,C 0.1093,E1 10.2281,E2 296.1413} C_DIS
LIN {X -123.0729,Y 56.2507,Z 168,A 156.3978,B 10.3715,C 0.1148,E1 10.2263,E2 294.5846} C_DIS
LIN {X -124.6011,Y 52.7803,Z 168,A 158.1625,B 10.3715,C 0.1161,E1 10.2243,E2 292.8023} C_DIS
LIN {X -126.0574,Y 49.1966,Z 168,A 159.7975,B 10.3715,C 0.1206,E1 10.2226,E2 291.1694} C_DIS
LIN {X -127.5481,Y 45.197,Z 168,A 161.6775,B 10.3715,C 0.1243,E1 10.2208,E2 289.2826} C_DIS
LIN {X -128.8125,Y 41.4509,Z 168,A 163.2488,B 10.3714,C 0.1309,E1 10.2195,E2 287.7256} C_DIS
LIN {X -129.7884,Y 38.2858,Z 168,A 164.6389,B 10.3714,C 0.1351,E1 10.2183,E2 286.3386} C_DIS
LIN {X -130.6531,Y 35.2231,Z 168,A 166.073,B 10.3713,C 0.1373,E1 10.2173,E2 284.8954} C_DIS
LIN {X -131.5396,Y 31.7508,Z 168,A 167.4613,B 10.3712,C 0.144,E1 10.2163,E2 283.5244} C_DIS
LIN {X -132.2798,Y 28.5103,Z 168,A 168.9728,B 10.3712,C 0.1461,E1 10.2154,E2 282.0017} C_DIS
LIN {X -132.9635,Y 25.1312,Z 168,A 170.5304,B 10.3712,C 0.1485,E1 10.2146,E2 280.4338} C_DIS
LIN {X -133.8125,Y 20.1338,Z 168,A 172.6507,B 10.371,C 0.1552,E1 10.2136,E2 278.319} C_DIS
LIN {X -134.3308,Y 16.3137,Z 168,A 174.3689,B 10.371,C 0.1583,E1 10.213,E2 276.592} C_DIS
LIN {X -134.6905,Y 13.012,Z 168,A 175.7772,B 10.371,C 0.1624,E1 10.2126,E2 275.1848} C_DIS
LIN {X -134.9997,Y 9.2867,Z 168,A 177.4783,B 10.3709,C 0.1648,E1 10.2123,E2 273.471} C_DIS
LIN {X -135.2165,Y 5.2309,Z 168,A 179.1338,B 10.3708,C 0.171,E1 10.2121,E2 271.825} C_DIS
LIN {X -135.3152,Y 0.9659,Z 168,A -179.0668,B 10.3707,C 0.1764,E1 10.212,E2 270.0283} C_DIS
LIN {X -135.2862,Y -3.0104,Z 168,A -177.1975,B 10.3707,C 0.1778,E1 10.212,E2 268.138} C_DIS
LIN {X -135.1281,Y -7.1681,Z 168,A -175.4402,B 10.3706,C 0.183,E1 10.2123,E2 266.3829} C_DIS
Enddeposition()
END
